   // Загружаем текущие флаги состояния
   #dm := #Bm;
   #Dx := #Bm;
   // Сбрасываем флаг первого цикла
   #Fx.Res := 0;
   // Назначаем группу сообщений (механизмов)
   // NDEV.GRP := SEL(G := 0 = #GRP, IN0 := #GRP, IN1 := PDEV.GRP);
   // Получаем структуру состояния привода
   IF (#Md.PZD) THEN
       #RRD := DPRD_DAT(LADDR := #LA, RECORD => #iT352);
   ELSE
       #RRD := DPRD_DAT(LADDR := #LA, RECORD => #iP6);
   END_IF;
   // Обрабатываем (непрерывные) данные состояния привода
   #SW := #SWx;
   #Re.X.SW := #SW;
   #Vx := #iT352.PZD2 / 16384.0 * #Vn;
   #Re.X.Vx := #Vx;
   #Ix := #iT352.PZD3 / 163.84;
   #Re.X.Ix := #Ix;
   #Mx := #iT352.PZD4 / 163.84;
   #Re.X.Mx := #Mx;
   #An := #iT352.PZD5;
   #Re.X.An := #An;
   #Fn := #iT352.PZD6;
   #Re.X.Fn := #Fn;
   #Brk := #iT352.PZD1.b02;
   #Re.X.Brk := #Brk;
   #Flt := #iT352.PZD1.b03 OR (#DPx = 0);
   #Re.X.Err := #Flt;
   #Alm := #iT352.PZD1.b07;
   // Обрабатываем дополнительные данные
   #P7 := #iT352.PZD7;
   #P8 := #iT352.PZD8;
   #P9 := #iT352.PZD9;
   // Передача параметров Master=>Slave
   IF (#Re.S.Mst) THEN
       // Данный привод является основным
       #Re."M".UBr := #UBr;
       #Re."M".Enb := #Enb;
       #Re."M".KOn := #KOn;
       #Re."M".Run := #Run;
       #Re."M".Ack := #Ack  OR "_ACK";
       #Re."M".Id := #Id;
       #Re."M".Ms := #Ms;
       #Re."M".Vs := #Vs;
       #Re."M".Vn := #Vn;
   ELSE
       // Данный привод является резервным
       #UBr := #Re."M".UBr;
       #Enb := #Re."M".Enb;
       #KOn := #Re."M".KOn;
       #Run := #Re."M".Run;
       #Ack := #Re."M".Ack;
       #Id := #Re."M".Id;
       #Ms := #Re."M".Ms;
       #Vs := #Re."M".Vs;
       #Vn := #Re."M".Vn;
   END_IF;
   // Формируем признаки устройства ввода резерва
   #Rd1 := #Re.S.Rd1;
   #SF.Rd1 := #Re.S.Rd1;
   #Rd2 := #Re.S.Rd2;
   #SF.Rd2 := #Re.S.Rd2;
   // Обработка состояния моторного модуля
   #SF.Flt := #Flt;
   #Fx.Flt := #Flt;
   #SF.Alm := #Alm;
   #Fx.Alm := #Alm;
   // Фиксируем текущие флаги
   #Fx.Mse :=  #Mse;               // (#PDEV.Msd = 0) &      // Разрешение выдачи сообщений для HMI
   #Fx.EnF := #Fx.Mse & #Md.EnF;                        // Разрешено сообщение Fault (отказ)
   #Fx.MsF := (#Fn <> 0) & #Fx.EnF;                        // Наличие сообщения Fault (отказ)
   #Fx.EnA := #Fx.Mse & #Md.EnA;                        // Разрешено сообщение Alarm (предупреждение)
   #Fx.MsA := (#An <> 0) & #Fx.EnA;                        // Наличие сообщения Alarm (предупреждение)
   #Fx.Rdy := #iT352.PZD1.b00;                         // Сигнал готовности привода (b00)
   #Fx.KOn := (#KOn OR #Run) & ((#Md.Rst = 0) OR #Fx.Rdy);  // Включить привод KOn|Run (команда)
   // Обрабатываем таймеры изменения состояния
   IF (#Fx.Tx0 OR #Fx.Tx1) THEN
       #Fx.Tx1 := ("_Time" - #Tm1 < #Ts1) & #Fx.Tx1;
       #Fx.Tx0 := ("_Time" - #Tm0 < #Md.Ts0) & #Fx.Tx0 & #Rdy & #Enb & (#Flt = 0);
   END_IF;
   // Фиксируем наличие событий
   #Dp := #Dx XOR #dm;
   // Обработка событий
   //  *** IF (#Dp <> 0) THEN
       // Запрос на инициализацию данных
   IF (#Fm.Res) THEN
           // Устанавливаем номер данного Instance Data Block
         (*#NDEV.IDB := 123; //- GetDINO();
           // Назначаем общие параметры сообщения
           #ME.Pr.N2 := #NDEV.IDB; *)
           // Инициализация данных
           #ME.Pr.N2 := 0;
           #ME.Pr.N4 := 0;
           #ME.Pr.N5 := 0;
           // Устанавливаем номер данного Instance Data Block
           #TPA := #ME;
           #NDB := #TSA.PTR.DN;
           // Назначаем группу сообщений (механизмов)
           IF (#GRP = 0) THEN
               #GRP := #NDB * 100;
           END_IF;
       END_IF;
       // Производим контроль изменения Rdy
       IF (#Fp.Rdy) THEN
           #Fx.Tx1 := (#Ts1 > T#0s) & #Fm.Rdy;
           #Tm1 := "_Time";
       END_IF;
       #Fx.Tx1 := (#Flt = 0) & #Fx.Tx1;
       #Rdy := #Fx.Tx1 OR #Fx.Rdy;
       #Re.X.Rdy := #Rdy;
       // Производим контроль изменения KOn
       IF (#Fp.KOn) THEN
           #Fx.Tx0 := (#Md.Ts0 > T#0s) & #Fm.KOn;
           #Tm0 := "_Time";
       END_IF;
       #Fx.Tx0 := (#Flt = 0) & #Fx.Tx0;
       #Fx.Run := #Fx.KOn OR #Fx.Tx0;
       // Устанавливаем активность сообщения Alarm (предупреждение)
       IF (#Fp.MsA XOR #MsAlm.SIG) THEN
           // Назначаем группу сообщений (механизмов)
           // Запрос на инициализацию данных
           #ME.Pr.N1 := #GRP;
           #ME.Pr.N2.%X0 := #Fm.MsA;
           #ME.Pr.N4 := 13;
           #ME.Pr.N6 := #GRP + 1;
           #MsAlm(SIG := (#Fp.MsA),
                  TIMESTAMP := "TS0",
                  SD_1 := #ME.Pr.N1,
                  SD_2 := #ME.Pr.N2,
                  SD_4 := #ME.Pr.N4,
                  SD_6 := #ME.Pr.N6);
       END_IF;
       // Устанавливаем активность сообщения Fault (отказ)
       IF (#Fp.MsF XOR #MsFlt.SIG)  THEN
          // Назначаем группу сообщений (механизмов)
          // Запрос на инициализацию данных
           #ME.Pr.N1 := #GRP;
           #ME.Pr.N2.%X0 := #Fm.MsF;
           #ME.Pr.N6 := #GRP + 2;
           #MsFlt(SIG := (#Fp.MsF),
                  TIMESTAMP := "TS0",
                  SD_1 := #ME.Pr.N1,
                  SD_2 := #ME.Pr.N2,
                  SD_6 := #ME.Pr.N6);
       END_IF;

       // Сохраняем текущее значение флагов
       #Bm := #Dx;
       //  *** END_IF;
   // Подготовка управляющей структуры привода
   #qT352.PZD1.b00 := ((#Re.S.Mst = 0) & #Re.S.Rd2 OR #Re.S.Mst & #Re.S.Rd1) & #Fx.Run;
   #qT352.PZD1.b02 := (#Re.S.Dis = 0) & #Enb & #DPx;
   #qT352.PZD1.b07 := #Re."M".Ack OR "_ACK";
   #qT352.PZD1.b12 := #UBr;
   // Обработка уставки скорости
   IF (#Run) THEN
       // Режим работы со скоростью и моментом
       #Vm := ABS(#Vn * 1.95);
       #Vs := LIMIT(MN := - #Vm, IN := #Vs, MX := + #Vm);
       #qT352.PZD2 := DINT_TO_INT(ROUND(#Vs / #Vn * 16384.0));
   ELSE
       // Режим намагничивания
       #qT352.PZD2 := 0;
   END_IF;
   // Обработка уставки момента
   IF (#Run OR #KOn) THEN
       #Ms := LIMIT(MN := -195.0, IN := #Ms, MX := +195.0);
       #qT352.PZD3 := DINT_TO_INT(ROUND(#Ms * 163.84));
   ELSE
       #qT352.PZD3 := 0;
   END_IF;
   // Формируем дополнительный параметр
   #qT352.PZD4 := #Id;
   // Передаем структуру управления привода
   IF (#Md.PZD) THEN
        #RWR := DPWR_DAT(LADDR := #LA, RECORD := #qT352);
   ELSE
        #RWR := DPWR_DAT(LADDR := #LA, RECORD := #qP6);
   END_IF;
   // Сбрасываем признак запрета
   #Re.S.Dis := 0;
   // Формируем индикацию для HMI
   #SF.Rdy := #Rdy;
   #SF.Qm0 := 0;
   #SF.Qm1 := #Re.S.Mst;
   #SF.Qm2 := #SF.Qm1 = 0;
END_FUNCTION_BLOCK

(* ===== HMI "HMI_RT_1" =====
system functions are stored by id; their names below are inferred from use
connection "HMI_Connection_1": ETHERNET, S7_1500_OMS

HMI tags "Default tag table"
   "Tag_ScreenNumber" : UInt, internal
   "AiCh_TE7.1_Px" : Real = PLC "AiCh_TE7.1".Px AT %DB7.DBD50, 1 s
   "AiCh_TE7.2_Px" : Real = PLC "AiCh_TE7.2".Px AT %DB8.DBD50, 1 s
   "Data_LevelVO_Pv" : Real = PLC Data.LevelVO_Pv, 1 s
   "DriveM7_1_Vx" : Real = PLC DriveM7_1.Vx AT %DB34.DBD78, 1 s
   "DriveM7_2_Vx" : Real = PLC DriveM7_2.Vx AT %DB35.DBD78, 1 s
   "AiCh_TE1.1_Px" : Real = PLC "AiCh_TE1.1".Px AT %DB1.DBD50, 1 s
   "AiCh_TE1.3_Px" : Real = PLC "AiCh_TE1.3".Px AT %DB3.DBD50, 1 s
   "AiCh_TE1.2_Px" : Real = PLC "AiCh_TE1.2".Px AT %DB2.DBD50, 1 s
   "DriveM1_1_Vx" : Real = PLC DriveM1_1.Vx AT %DB33.DBD78, 1 s
   "AiCh_LIC1.1_Px" : Real = PLC "AiCh_LIC1.1".Px AT %DB12.DBD50, 1 s
   "AiCh_TE2.1_Px" : Real = PLC "AiCh_TE2.1".Px AT %DB4.DBD50, 1 s
   "AiCh_TE2.3_Px" : Real = PLC "AiCh_TE2.3".Px AT %DB6.DBD50, 1 s
   "AiCh_TE2.2_Px" : Real = PLC "AiCh_TE2.2".Px AT %DB5.DBD50, 1 s
   "DriveM2_1_Vx" : Real = PLC DriveM2_1.Vx AT %DB38.DBD78, 1 s
   "AiCh_LIC2.1_Px" : Real = PLC "AiCh_LIC2.1".Px AT %DB13.DBD50, 1 s
   "Data_ACK" : Bool = PLC Data.Ack, 1 s
   "Data_MAN_ON" : Bool = PLC Data.MAN_ON, 1 s
   "Data_Reg_TE1_1_Sp" : Real = PLC Data.Reg_TE1_1.Sp, 1 s
   "Di_Lah1.1" : Bool = PLC "Di_Lah1.1" AT %I42.6, 1 s
   "Di_Ga1.4" : Bool = PLC "Di_Ga1.4" AT %I44.3, 1 s
   "DrvCell_M1_1_SB1" : Bool = PLC DrvCell_M1_1.SB1 AT %DB36.DBX16.0, 1 s
   "DrvCell_M1_1_Err" : Bool = PLC DrvCell_M1_1.Err AT %DB36.DBX74.1, 1 s
   "DrvCell_M1_1_Km1" : Bool = PLC DrvCell_M1_1.Km1 AT %DB36.DBX73.0, 1 s
   "DrvCell_M2_1_Err" : Bool = PLC DrvCell_M2_1.Err AT %DB37.DBX74.1, 1 s
   "DrvCell_M1_2_Km1" : Bool = PLC DrvCell_M1_2.Km1 AT %DB17.DBX73.0, 1 s
   "DrvCell_M1_2_Err" : Bool = PLC DrvCell_M1_2.Err AT %DB17.DBX74.1, 1 s
   "DrvCell_M1_2_SB1" : Bool = PLC DrvCell_M1_2.SB1 AT %DB17.DBX16.0, 1 s
   "DrvCell_V1_7_Err" : Bool = PLC DrvCell_V1_7.Err AT %DB28.DBX74.1, 1 s
   "DrvCell_V1_7_Km1" : Bool = PLC DrvCell_V1_7.Km1 AT %DB28.DBX73.0, 1 s
   "DrvCell_V1_7_SB1" : Bool = PLC DrvCell_V1_7.SB1 AT %DB28.DBX16.0, 1 s
   "Data_Mixer1_Direction" : Int = PLC Data.Mixer1.Direction, 1 s
   "Data_Equipment_Work" : Bool = PLC Data.Equipment_Work, 1 s
   "DrvCell_V1_1_SB1" : Bool = PLC DrvCell_V1_1.SB1 AT %DB25.DBX16.0, 1 s
   "DrvCell_V1_1_Err" : Bool = PLC DrvCell_V1_1.Err AT %DB25.DBX74.1, 1 s
   "DrvCell_M2_1_SB1" : Bool = PLC DrvCell_M2_1.SB1 AT %DB37.DBX16.0, 1 s
   "DrvCell_M2_1_Lr2" : Bool = PLC DrvCell_M2_1.Lr2 AT %DB37.DBX73.7, 1 s
   "DrvCell_M2_1_Km1" : Bool = PLC DrvCell_M2_1.Km1 AT %DB37.DBX73.0, 1 s
   "Data_Mixer2_Direction" : Int = PLC Data.Mixer2.Direction, 1 s
   "Di_Ga2.4" : Bool = PLC "Di_Ga2.4" AT %I44.7, 1 s
   "Data_Reg_TE2_1_Sp" : Real = PLC Data.Reg_TE2_1.Sp, 1 s
   "Di_Lah2.1" : Bool = PLC "Di_Lah2.1" AT %I42.7, 1 s
   "DrvCell_V2_1_SB1" : Bool = PLC DrvCell_V2_1.SB1 AT %DB26.DBX16.0, 1 s
   "DrvCell_V2_1_Err" : Bool = PLC DrvCell_V2_1.Err AT %DB26.DBX74.1, 1 s
   "DrvCell_V2_1_Km1" : Bool = PLC DrvCell_V2_1.Km1 AT %DB26.DBX73.0, 1 s
   "DrvCell_M2_2_SB1" : Bool = PLC DrvCell_M2_2.SB1 AT %DB18.DBX16.0, 1 s
   "DrvCell_M2_2_Err" : Bool = PLC DrvCell_M2_2.Err AT %DB18.DBX74.1, 1 s
   "DrvCell_M2_2_Km1" : Bool = PLC DrvCell_M2_2.Km1 AT %DB18.DBX73.0, 1 s
   "DrvCell_V2_7_SB1" : Bool = PLC DrvCell_V2_7.SB1 AT %DB29.DBX16.0, 1 s
   "DrvCell_V2_7_Err" : Bool = PLC DrvCell_V2_7.Err AT %DB29.DBX74.1, 1 s
   "DrvCell_V2_7_Km1" : Bool = PLC DrvCell_V2_7.Km1 AT %DB29.DBX73.0, 1 s
   "DrvCell_V1_1_Km1" : Bool = PLC DrvCell_V1_1.Km1 AT %DB25.DBX73.0, 1 s
   "Data_Mixer1_Man" : Real = PLC Data.Mixer1.Man, 1 s
   "Data_Mixer2_Man" : Real = PLC Data.Mixer2.Man, 1 s
   "Di_Ga1.1" : Bool = PLC "Di_Ga1.1" AT %I44.0, 1 s
   "Di_Ga1.2" : Bool = PLC "Di_Ga1.2" AT %I44.1, 1 s
   "Di_Ga2.1" : Bool = PLC "Di_Ga2.1" AT %I44.4, 1 s
   "Di_Ga2.2" : Bool = PLC "Di_Ga2.2" AT %I44.5, 1 s
   "DrvCell_M5_SB1" : Bool = PLC DrvCell_M5.SB1 AT %DB59.DBX16.0, 1 s
   "DrvCell_M5_Err" : Bool = PLC DrvCell_M5.Err AT %DB59.DBX74.1, 1 s
   "DrvCell_M5_Km1" : Bool = PLC DrvCell_M5.Km1 AT %DB59.DBX73.0, 1 s
   "DrvCell_M4_Err" : Bool = PLC DrvCell_M4.Err AT %DB21.DBX74.1, 1 s
   "DrvCell_M4_Km1" : Bool = PLC DrvCell_M4.Km1 AT %DB21.DBX73.0, 1 s
   "DrvCell_M4_SB1" : Bool = PLC DrvCell_M4.SB1 AT %DB21.DBX16.0, 1 s
   "Di_1Ga06" : Bool = PLC Di_1Ga06 AT %I46.4, 1 s
   "Di_1Ga01" : Bool = PLC Di_1Ga01 AT %I45.6, 1 s
   "Di_1Ga02" : Bool = PLC Di_1Ga02 AT %I46.0, 1 s
   "Data_Kr1_TempFilling" : Real = PLC Data.Kr1.TempFilling, 1 s
   "Data_Kr1_TempKristal" : Real = PLC Data.Kr1.TempKristal, 1 s
   "Kr_1_Work_Run" : Bool = PLC Kr_1_Work.Run, 1 s
   "Data_Kr1_TimeKristal" : Int = PLC Data.Kr1.TimeKristal, 1 s
   "Kr_1_Work_LeftTimeMin" : DInt = PLC Kr_1_Work.LeftTimeMin, 1 s
   "Data_Kr1_Regim" : Int = PLC Data.Kr1.Regim, 1 s
   "Data_Kr1_Start" : Bool = PLC Data.Kr1.Start, 1 s
   "Data_Kr1_Stop" : Bool = PLC Data.Kr1.Stop, 1 s
   "Data_Mixer1_Power" : Real = PLC Data.Mixer1.Power, 1 s
   "Data_Mixer1_TimeRight" : DInt = PLC Data.Mixer1.TimeRight, 1 s
   "Data_Mixer1_TimeLeft" : DInt = PLC Data.Mixer1.TimeLeft, 1 s
   "Data_Mixer1_TimePause" : DInt = PLC Data.Mixer1.TimePause, 1 s
   "Data_Mixer1_RegimBothSide" : Bool = PLC Data.Mixer1.RegimBothSide, 1 s
   "Data_Mixer1_Start" : Bool = PLC Data.Mixer1.Start, 1 s
   "Data_Mixer1_Stop" : Bool = PLC Data.Mixer1.Stop, 1 s
   "Data_Kr1_Ready_Work" : Bool = PLC Data.Kr1.Ready_Work, 1 s
   "Data_Kr1_Ready_Route" : Bool = PLC Data.Kr1.Ready_Route, 1 s
   "Data_GlobalErrorStop" : Bool = PLC Data.GlobalErrorStop, 1 s
   "Data_Kr2_TempFilling" : Real = PLC Data.Kr2.TempFilling, 1 s
   "Kr_2_Work_Run" : Bool = PLC Kr_2_Work.Run, 1 s
   "Data_Kr2_TempKristal" : Real = PLC Data.Kr2.TempKristal, 1 s
   "Data_Kr2_TimeKristal" : Int = PLC Data.Kr2.TimeKristal, 1 s
   "Kr_2_Work_LeftTimeMin" : DInt = PLC Kr_2_Work.LeftTimeMin, 1 s
   "Data_Kr2_Regim" : Int = PLC Data.Kr2.Regim, 1 s
   "Data_Kr2_Start" : Bool = PLC Data.Kr2.Start, 1 s
   "Data_Kr2_Stop" : Bool = PLC Data.Kr2.Stop, 1 s
   "Data_Kr2_Ready_Work" : Bool = PLC Data.Kr2.Ready_Work, 1 s
   "Data_Kr2_Ready_Route" : Bool = PLC Data.Kr2.Ready_Route, 1 s
   "Data_Mixer2_Power" : Real = PLC Data.Mixer2.Power, 1 s
   "Data_Mixer2_TimeRight" : DInt = PLC Data.Mixer2.TimeRight, 1 s
   "Data_Mixer2_TimeLeft" : DInt = PLC Data.Mixer2.TimeLeft, 1 s
   "Data_Mixer2_TimePause" : DInt = PLC Data.Mixer2.TimePause, 1 s
   "Data_Mixer2_RegimBothSide" : Bool = PLC Data.Mixer2.RegimBothSide, 1 s
   "Data_Mixer2_Start" : Bool = PLC Data.Mixer2.Start, 1 s
   "Data_Mixer2_Stop" : Bool = PLC Data.Mixer2.Stop, 1 s
   "Data_washing_cipRegim" : Int = PLC Data.washing.cipRegim, 1 s
   "Data_washing_Start" : Bool = PLC Data.washing.Start, 1 s
   "Data_washing_Stop" : Bool = PLC Data.washing.Stop, 1 s
   "Data_washing_readyGlobal" : Bool = PLC Data.washing.readyGlobal, 1 s
   "Data_washing_readyRoute" : Bool = PLC Data.washing.readyRoute, 1 s
   "WashingWork_DB_Run" : Bool = PLC WashingWork_DB.Run, 1 s
   "Data_Reg_M7_1_Sp" : Real = PLC Data.Reg_M7_1.Sp, 1 s
   "Data_Reg_01RV01_Sp" : Real = PLC Data.Reg_01RV01.Sp, 1 s
   "Data_Power_7_2" : Real = PLC Data.Power_7_2, 1 s
   "Kr_1_Work_Step" : Int = PLC Kr_1_Work.Step, 1 s
   "Kr_2_Work_Step" : Int = PLC Kr_2_Work.Step, 1 s
   "Data_GlobalError" : Bool = PLC Data.GlobalError, 1 s
   "DrvCell_V7_3_Err" : Bool = PLC DrvCell_V7_3.Err AT %DB31.DBX74.1, 1 s
   "DrvCell_V7_3_Km1" : Bool = PLC DrvCell_V7_3.Km1 AT %DB31.DBX73.0, 1 s
   "DrvCell_V7_4_Err" : Bool = PLC DrvCell_V7_4.Err AT %DB32.DBX74.1, 1 s
   "DrvCell_V7_4_Km1" : Bool = PLC DrvCell_V7_4.Km1 AT %DB32.DBX73.0, 1 s
   "DrvCell_V7_3_SB1" : Bool = PLC DrvCell_V7_3.SB1 AT %DB31.DBX16.0, 1 s
   "DrvCell_V7_4_SB1" : Bool = PLC DrvCell_V7_4.SB1 AT %DB32.DBX16.0, 1 s
   "Data_Reg_01RV01_LMN" : Real = PLC Data.Reg_01RV01.LMN, 1 s
   "Data_Reg_01RV01_Man" : Real = PLC Data.Reg_01RV01.Man, 1 s
   "DrvCell_V7_1_Err" : Bool = PLC DrvCell_V7_1.Err AT %DB23.DBX74.1, 1 s
   "DrvCell_V7_1_Km1" : Bool = PLC DrvCell_V7_1.Km1 AT %DB23.DBX73.0, 1 s
   "DrvCell_V7_1_SB1" : Bool = PLC DrvCell_V7_1.SB1 AT %DB23.DBX16.0, 1 s
   "DrvCell_M7_1_Err" : Bool = PLC DrvCell_M7_1.Err AT %DB39.DBX74.1, 1 s
   "DrvCell_M7_1_Km1" : Bool = PLC DrvCell_M7_1.Km1 AT %DB39.DBX73.0, 1 s
   "DrvCell_M7_1_SB1" : Bool = PLC DrvCell_M7_1.SB1 AT %DB39.DBX16.0, 1 s
   "Data_Reg_M7_1_Man" : Real = PLC Data.Reg_M7_1.Man, 1 s
   "DrvCell_M10_Err" : Bool = PLC DrvCell_M10.Err AT %DB22.DBX74.1, 1 s
   "DrvCell_M10_Km1" : Bool = PLC DrvCell_M10.Km1 AT %DB22.DBX73.0, 1 s
   "DrvCell_M10_SB1" : Bool = PLC DrvCell_M10.SB1 AT %DB22.DBX16.0, 1 s
   "DrvCell_M3_Err" : Bool = PLC DrvCell_M3.Err AT %DB20.DBX74.1, 1 s
   "DrvCell_M3_Km1" : Bool = PLC DrvCell_M3.Km1 AT %DB20.DBX73.0, 1 s
   "DrvCell_M3_SB1" : Bool = PLC DrvCell_M3.SB1 AT %DB20.DBX16.0, 1 s
   "Di_Lah01" : Bool = PLC Di_Lah01 AT %I43.1, 1 s
   "Di_Lal01" : Bool = PLC Di_Lal01 AT %I43.2, 1 s
   "DrvCell_M7_2_Err" : Bool = PLC DrvCell_M7_2.Err AT %DB40.DBX74.1, 1 s
   "DrvCell_M7_2_Km1" : Bool = PLC DrvCell_M7_2.Km1 AT %DB40.DBX73.0, 1 s
   "DrvCell_M7_2_SB1" : Bool = PLC DrvCell_M7_2.SB1 AT %DB40.DBX16.0, 1 s
   "Data_Reg_M7_2_Man" : Real = PLC Data.Reg_M7_2.Man, 1 s
   "DrvCell_V7_2_SB1" : Bool = PLC DrvCell_V7_2.SB1 AT %DB24.DBX16.0, 1 s
   "DrvCell_V7_2_Err" : Bool = PLC DrvCell_V7_2.Err AT %DB24.DBX74.1, 1 s
   "DrvCell_V7_2_Km1" : Bool = PLC DrvCell_V7_2.Km1 AT %DB24.DBX73.0, 1 s
   "ViewLine_DB_Line2" : Int = PLC ViewLine_DB.Line2, 1 s
   "ViewLine_DB_Line1" : Int = PLC ViewLine_DB.Line1, 1 s
   "ViewLine_DB_Line3" : Int = PLC ViewLine_DB.Line3, 1 s
   "ViewLine_DB_Line4" : Int = PLC ViewLine_DB.Line4, 1 s
   "ViewLine_DB_Line5" : Int = PLC ViewLine_DB.Line5, 1 s
   "ViewLine_DB_Line7" : Int = PLC ViewLine_DB.Line7, 1 s
   "ViewLine_DB_Line8" : Int = PLC ViewLine_DB.Line8, 1 s
   "ViewLine_DB_Line9" : Int = PLC ViewLine_DB.Line9, 1 s
   "ViewLine_DB_Line10" : Int = PLC ViewLine_DB.Line10, 1 s
   "ViewLine_DB_Line11" : Int = PLC ViewLine_DB.Line11, 1 s
   "ViewLine_DB_Line12" : Int = PLC ViewLine_DB.Line12, 1 s
   "Messages" : Word AT %DB44.DBW0, 1 s
   "ViewLine_DB_Line13" : Int = PLC ViewLine_DB.Line13, 1 s
   "ViewLine_DB_Line14" : Int = PLC ViewLine_DB.Line14, 1 s
   "ViewLine_DB_Line17" : Int = PLC ViewLine_DB.Line17, 1 s
   "ViewLine_DB_Line15" : Int = PLC ViewLine_DB.Line15, 1 s
   "ViewLine_DB_Line16" : Int = PLC ViewLine_DB.Line16, 1 s
   "ViewLine_DB_Line25" : Int = PLC ViewLine_DB.Line25, 1 s
   "ViewLine_DB_Line24" : Int = PLC ViewLine_DB.Line24, 1 s
   "ViewLine_DB_Line23" : Int = PLC ViewLine_DB.Line23, 1 s
   "ViewLine_DB_Line18" : Int = PLC ViewLine_DB.Line18, 1 s
   "ViewLine_DB_Line19" : Int = PLC ViewLine_DB.Line19, 1 s
   "ViewLine_DB_Line20" : Int = PLC ViewLine_DB.Line20, 1 s
   "ViewLine_DB_Line21" : Int = PLC ViewLine_DB.Line21, 1 s
   "ViewLine_DB_Line22" : Int = PLC ViewLine_DB.Line22, 1 s
   "WashingWork_DB_Step" : Int = PLC WashingWork_DB.Step, 1 s
   "Data_ReadyKr1" : Bool = PLC Data.ReadyKr1, 1 s
   "Data_Power_7_2_CIP" : Real = PLC Data.Power_7_2_CIP, 1 s
   "Data_EnableReady" : Bool = PLC Data.EnableReady, 1 s
   "Data_ReadyKr2" : Bool = PLC Data.ReadyKr2, 1 s
   "Data_ReadyCIP" : Bool = PLC Data.ReadyCIP, 1 s

discrete alarms
   11: 'Нажата аварийная кнопка', class Errors, trigger "Messages" bit 8
   12: 'Напряжение 380В не в норме', class Errors, trigger "Messages" bit 9
   13: 'Нет давления воздуха в пневмосистеме', class Errors, trigger "Messages" bit 10
   14: 'Верхний аварийный уровень кристализатора №1', class Errors, trigger "Messages" bit 11
   15: 'Верхний аварийный уровень кристализатора №2', class Errors, trigger "Messages" bit 12
   16: 'Верхний аварийный уровень емкости ледянной воды', class Errors, trigger "Messages" bit 13
   17: 'UPS, батарея разряжена', class Warnings, trigger "Messages" bit 14
   18: 'UPS, батарея неисправна', class No Acknowledgement, trigger "Messages" bit 15
   19: 'Открыт люк 1 кристализатора', class Errors, trigger "Messages" bit 0
   20: 'Открыт люк 2 кристализатора', class Errors, trigger "Messages" bit 1

text list "Kristal_Regim": 1 'Наполнение'; 2 'Кристализация'; 3 'Выкачка'

text list "cipRegim": 1 'Мойка линии подачи продукта'; 2 'Мойка линии выгрузки продукта'; 3 'Мойка кристализатора №1'; 4 'Мойка кристализатора №2'

text list "on/off": 0 'Отключено'; 1 'Включено'

Template "Template_1" 800x434
   Button "Template_Button_9" at 2,375 size 100x58; TextOff 'Вакуумный охладитель'
      on Release: ActivateScreen("mainVo", 0)
   AlarmView "Alarm view_Unacknowledged" at 0,357 size 800x19
   Button "Template_Button_5" at 104,375 size 100x58; TextOff 'Кристализа- торы'
      on Release: ActivateScreen("Kristals", 0)
   Button "Template_Button_6" at 406,375 size 96x58; TextOff 'Сообщения'
      on Release: ActivateScreen("messages", 0)
   Button "Template_Button_3" at 504,375 size 96x58; TextOff 'Настройки'
      on Release: ActivateScreen("SettingsCommon", 0)
   Button "Template_Button_4" at 206,375 size 100x58; TextOff 'Линии крист.'
      on Release: ActivateScreen("Lines", 0)
   Button "Template_Button_7" at 308,375 size 96x58; TextOff 'Графики'
      on Release: ActivateScreen("TrendsCommon", 0)
   Button "Template_Button_1" at 602,375 size 96x58; TextOff 'Сброс аварии'
      on Press: function_b14e0dd5("Data_ACK", 0)
   Button "Template_Button_2" at 700,375 size 96x58; TextOff 'Ручной'
      on Press: InvertBit("Data_MAN_ON")
      Appearance <- "Data_MAN_ON"
      ObjectEnable <- "Data_Equipment_Work"

screen "mainVo" 800x434, template "Template_1"
   on GenerateScreen: SetTag("Tag_ScreenNumber", 1)
   Rectangle "Rectangle_12" at 233,159 size 68x24; ToolTipText 'Температура НС'
   TextField "Text field_15" at 274,159 size 18x22; Text '%'
   IOField "IO Field_11" at 236,157 size 36x26; FormatPattern 999
      ProcessValue <- "Data_LevelVO_Pv"
   SymbolLibrary "Symbol library_35" at 261,235 size 13x60
      Appearance <- "ViewLine_DB_Line1"
   SymbolLibrary "Symbol library_56" at 167,48 size 13x149
      Appearance <- "ViewLine_DB_Line2"
   SymbolLibrary "Symbol library_1" at 63,195 size 166x13
      Appearance <- "ViewLine_DB_Line1"
   SymbolLibrary "Symbol library_6" at 255,12 size 54x54
   SymbolLibrary "Symbol library_9" at 217,28 size 25x25
      Appearance <- "ViewLine_DB_Line2"
   SymbolLibrary "Symbol library_4" at 219,39 size 98x199
   SymbolLibrary "Symbol library_31" at 714,259 size 13x43
      Appearance <- "DrvCell_M3_Km1"
   SymbolLibrary "Symbol library_160" at 714,143 size 13x49
   GraphicView "Graphic view_4" at 672,168 size 102x103; Picture "Graphic_5"
   SymbolLibrary "Symbol library_19" at 61,280 size 196x13
      Appearance <- "ViewLine_DB_Line7"
   SymbolLibrary "Symbol library_11" at 358,196 size 13x78
      Appearance <- "ViewLine_DB_Line7"
   SymbolLibrary "Symbol library_15" at 386,256 size 25x25
      Appearance <- "ViewLine_DB_Line3"
   SymbolLibrary "Symbol library_13" at 346,268 size 25x25
      Appearance <- "ViewLine_DB_Line7"
   Bar "Bar_1" at 223,67 size 90x143; MinimumValue 0; MaximumValue 100
      ProcessValue <- "Data_LevelVO_Pv"
   SymbolLibrary "Symbol library_7" at 307,12 size 55x28
   SymbolLibrary "Symbol library_2" at 188,28 size 37x13
      Appearance <- "ViewLine_DB_Line2"
   Group "Group_19" at 233,157 size 68x26
   SymbolLibrary "Symbol library_53" at 40,40 size 13x147
      Appearance <- "ViewLine_DB_Line1"
   SymbolLibrary "Symbol library_51" at 167,28 size 25x25
      Appearance <- "ViewLine_DB_Line2"
   SymbolLibrary "Symbol library_5" at 40,183 size 25x25
      Appearance <- "ViewLine_DB_Line1"
   SymbolLibrary "Symbol library_12" at 261,290 size 25x25
      Appearance <- "ViewLine_DB_Line1"
   SymbolLibrary "Symbol library_14" at 400,256 size 169x13
      Appearance <- "ViewLine_DB_Line3"
   SymbolLibrary "Symbol library_16" at 562,252 size 41x21
   SymbolLibrary "Symbol library_17" at 384,197 size 116x13
      Appearance <- "ViewLine_DB_Line5"
   SymbolLibrary "Symbol library_18" at 285,302 size 100x13
      Appearance <- "ViewLine_DB_Line1"
   SymbolLibrary "Symbol library_22" at 38,280 size 25x25
      Appearance <- "ViewLine_DB_Line7"
   SymbolLibrary "Symbol library_23" at 384,105 size 128x13
      Appearance <- "ViewLine_DB_Line4"
   SymbolLibrary "Symbol library_24" at 279,280 size 69x13
      Appearance <- "ViewLine_DB_Line7"
   SymbolLibrary "Symbol library_25" at 553,184 size 34x13
      Appearance <- "ViewLine_DB_Line5"
   TextField "Text field_2" at 592,205 size 23x43; Text 'Y'
   SymbolLibrary "Symbol library_29" at 507,67 size 25x25
      Appearance <- "ViewLine_DB_Line4"
   SymbolLibrary "Symbol library_30" at 585,184 size 25x25
      Appearance <- "ViewLine_DB_Line5"
   Circle "Circle_27" at 742,239 size 25x25
      Appearance <- "Di_Lal01"
   SymbolLibrary "Symbol library_36" at 702,299 size 25x25
      Appearance <- "DrvCell_M3_Km1"
   SymbolLibrary "Symbol library_34" at 613,296 size 61x13
      Appearance <- "DrvCell_M3_Km1"
   SymbolLibrary "Symbol library_161" at 591,292 size 25x21
   SymbolLibrary "Symbol library_37" at 710,122 size 21x25
   SymbolLibrary "Symbol library_27" at 531,67 size 113x13
      Appearance <- "ViewLine_DB_Line4"
   TextField "Static Text47_1" at 74,77 size 33x16; Text 'TE7.1 / TE04.1'
   Group "Group_17" at 49,91 size 82x26; FormatPattern 999.9
   SymbolLibrary "Symbol library_41" at 36,9 size 21x41
   TextField "Static Text47_2" at 176,213 size 33x16; Text 'TE7.2 / TE04.1'
   Group "Group_1" at 151,252 size 82x26; FormatPattern 999.9
   Group "Group_20" at 94,301 size 55x20; FormatPattern 999
   Group "Group_2" at 462,322 size 55x20; FormatPattern 999
   IOField "IO Field_12" at 36,243 size 47x31; FormatPattern 999
      Visibility <- "Data_MAN_ON"
      ProcessValue <- "Data_Reg_01RV01_Man"
   IOField "IO Field_2" at 466,287 size 47x31; FormatPattern 999
      Visibility <- "Data_MAN_ON"
      ProcessValue <- "Data_Reg_M7_1_Man"
   SymbolLibrary "Symbol library_20" at 258,340 size 108x7
      Appearance <- "ViewLine_DB_Line8"
   SymbolLibrary "Symbol library_42" at 241,336 size 30x15
   SymbolLibrary "Symbol library_44" at 362,334 size 15x13
      Appearance <- "ViewLine_DB_Line8"
   SymbolLibrary "Symbol library_43" at 369,316 size 15x13
      Appearance <- "ViewLine_DB_Line8"
   SymbolLibrary "Symbol library_45" at 412,143 size 81x7
      Appearance <- "ViewLine_DB_Line9"
   SymbolLibrary "Symbol library_47" at 400,138 size 30x15
   SymbolLibrary "Symbol library_49" at 490,137 size 11x13
      Appearance <- "ViewLine_DB_Line9"
   SymbolLibrary "Symbol library_50" at 494,118 size 12x13
      Appearance <- "ViewLine_DB_Line9"
   Group "Group_3" at 566,131 size 55x20; FormatPattern 999
   IOField "IO Field_3" at 570,92 size 47x31; FormatPattern 999
      Visibility <- "Data_MAN_ON"
      ProcessValue <- "Data_Reg_M7_2_Man"
   TextField "Text field_6" at 32,302 size 23x43; Text 'Y'
   TextField "Text field_7" at 647,87 size 23x43; Text 'Y'
   SymbolLibrary "Symbol library_28" at 640,67 size 25x25
      Appearance <- "ViewLine_DB_Line4"
   SymbolLibrary "Symbol library_38" at 494,130 size 7x14
      Appearance <- "ViewLine_DB_Line9"
   TextField "Static Text47_13" at 513,165 size 24x16; Text 'M10 / TE04.1'
   TextField "Static Text47_3" at 109,152 size 26x16; Text 'V7.3 / TE04.1'
   TextField "Static Text47_4" at 186,66 size 26x16; Text 'V7.4 / TE04.1'
   TextField "Static Text47_5" at 527,81 size 28x16; Text 'M7.2 / TE04.1'
   TextField "Static Text47_6" at 424,120 size 26x16; Text 'V7.2 / TE04.1'
   TextField "Static Text47_7" at 310,314 size 26x16; Text 'V7.1 / TE04.1'
   TextField "Static Text47_8" at 419,271 size 28x16; Text 'M7.1 / TE04.1'
   TextField "Static Text47_9" at 668,276 size 17x16; Text 'M3 / TE04.1'
   TextField "Static Text58_6" at 685,203 size 76x32; Text 'Ледянная вода RV01'
   Circle "Circle_26" at 742,176 size 25x25
      Appearance <- "Di_Lah01"
   ScreenModuleView "V7_31_1" at 105,169 size 43x40; ScreenModuleType ""
      Guid_{11997190-20001} <- "DrvCell_V7_3_Err"
      Guid_{11997190-19997} <- "DrvCell_V7_3_Km1"
   ScreenModuleView "M1_2_1" at 497,181 size 57x45; ScreenModuleType ""
      Guid_{11997190-21672} <- "DrvCell_M10_Err"
      Guid_{11997190-21676} <- "DrvCell_M10_Km1"
   ScreenModuleView "V1_7_1" at 308,330 size 30x25; ScreenModuleType ""
      Guid_{11997190-23352} <- "DrvCell_V7_1_Err"
      Guid_{11997190-23356} <- "DrvCell_V7_1_Km1"
   SymbolLibrary "Symbol library_3" at 341,8 size 44x222
   ScreenModuleView "RV01_2" at 87,234 size 51x64; ScreenModuleType ""
      Guid_{11997190-34850} <- "Data_Reg_01RV01_LMN"
   ScreenModuleView "М7_4_1" at 165,87 size 40x43; ScreenModuleType ""
      Guid_{11997190-20546} <- "DrvCell_V7_4_Err"
      Guid_{11997190-20554} <- "DrvCell_V7_4_Km1"
   Button "Button_6" at 85,148 size 73x73; TextOff 'Text'
      on Press: function_b14e0dd5("DrvCell_V7_3_SB1", 0)
   ScreenModuleView "M7_1_1" at 380,276 size 81x62; ScreenModuleType ""
      Guid_{11997190-20939} <- "DrvCell_M7_1_Err"
      Guid_{11997190-20935} <- "DrvCell_M7_1_Km1"
   Button "Button_7" at 374,242 size 88x113; TextOff 'Text'
      on Press: function_b14e0dd5("DrvCell_M7_1_SB1", 0)
   Button "Button_3" at 491,158 size 74x85; TextOff 'Text'
      on Press: function_b14e0dd5("DrvCell_M10_SB1", 0)
   ScreenModuleView "M_3_1" at 646,293 size 57x45; ScreenModuleType ""
      Guid_{11997190-24475} <- "DrvCell_M3_Err"
      Guid_{11997190-24471} <- "DrvCell_M3_Km1"
   Button "Button_8" at 637,271 size 74x85; TextOff 'Text'
      on Press: function_b14e0dd5("DrvCell_M3_SB1", 0)
   ScreenModuleView "V1_7_2" at 448,131 size 30x25; ScreenModuleType ""
      Guid_{11997190-23352} <- "DrvCell_V7_2_Err"
      Guid_{11997190-23356} <- "DrvCell_V7_2_Km1"
   ScreenModuleView "M7_21_1" at 504,91 size 59x53; ScreenModuleType ""
      Guid_{11997190-26153} <- "DrvCell_M7_2_Err"
      Guid_{11997190-26157} <- "DrvCell_M7_2_Km1"
   Group "Group_27" at 233,133 size 68x26
   Group "Group_4" at 151,228 size 82x26; FormatPattern 999.9
   Button "Button_1" at 494,67 size 74x85; TextOff 'Text'
      on Press: function_b14e0dd5("DrvCell_M7_2_SB1", 0)
   Button "Button_5" at 275,298 size 87x60; TextOff 'Text'
      on Press: function_b14e0dd5("DrvCell_V7_1_SB1", 0)
   Button "Button_2" at 414,115 size 74x53; TextOff 'Text'
      on Press: function_b14e0dd5("DrvCell_V7_2_SB1", 0)
   Button "Button_4" at 145,65 size 73x73; TextOff 'Text'
      on Press: function_b14e0dd5("DrvCell_V7_4_SB1", 0)
   SymbolLibrary "Symbol library_8" at 369,326 size 8x10
      Appearance <- "ViewLine_DB_Line8"
   Rectangle "Rectangle_1" at 56,93 size 75x24; ToolTipText 'Температура НС'
   TextField "Text field_3" at 106,93 size 19x22; Text 'С°'
   IOField "IO Field_10" at 49,91 size 56x26; FormatPattern 999.9
      ProcessValue <- "AiCh_TE7.1_Px"
   Rectangle "Rectangle_2" at 158,254 size 75x24; ToolTipText 'Температура НС'
   TextField "Text field_4" at 208,254 size 19x22; Text 'С°'
   IOField "IO Field_1" at 151,252 size 56x26; FormatPattern 999.9
      ProcessValue <- "AiCh_TE7.2_Px"
   IOField "I/O field_2" at 94,301 size 39x20; FormatPattern 999
      ProcessValue <- "Data_Reg_01RV01_LMN"
   TextField "Text field_16" at 130,302 size 19x19; Text '%'
   IOField "I/O field_1" at 462,322 size 39x20; FormatPattern 999
      ProcessValue <- "DriveM7_1_Vx"
   TextField "Text field_5" at 498,323 size 19x19; Text '%'
   IOField "I/O field_3" at 566,131 size 39x20; FormatPattern 999
      ProcessValue <- "DriveM7_2_Vx"
   TextField "Text field_1" at 602,132 size 19x19; Text '%'
   Rectangle "Rectangle_15" at 233,135 size 68x24; ToolTipText 'Температура НС'
   TextField "Text field_23" at 274,135 size 18x22; Text '%'
   IOField "IO Field_19" at 236,133 size 36x26; FormatPattern 999
      ProcessValue <- "Data_Reg_M7_1_Sp"
   Rectangle "Rectangle_3" at 158,230 size 75x24; ToolTipText 'Температура НС'
   TextField "Text field_8" at 208,230 size 19x22; Text 'С°'
   IOField "IO Field_4" at 151,228 size 56x26; FormatPattern 999.9
      ProcessValue <- "Data_Reg_01RV01_Sp"

screen "TrendsCommon" 800x434, template "Template_1"
   Button "Template_Button_7g" at 256,50 size 308x58; TextOff 'Вакуумохладитель'
      on Release: ActivateScreen("VO", 0)
   Button "Template_Button_8" at 256,109 size 308x58; TextOff 'Кристализатор №1'
      on Release: ActivateScreen("Kristalizator1", 0)
   Button "Template_Button_10" at 256,168 size 308x58; TextOff 'Кристализатор №2'
      on Release: ActivateScreen("Kristalizator2", 0)

screen "messages" 800x434, template "Template_1"
   AlarmView "Alarm view_1" at 0,2 size 798x321
   Button "Template_Button_5q" at 618,323 size 82x34; TextOff 'Архив'
      on Release: ActivateScreen("messagesArchive", 0)

screen "messagesArchive" 800x434, template "Template_1"
   AlarmView "Alarm view_1" at 0,0 size 798x356; AlarmLog "Alarm_log_1"

screen "VO" 800x434, template "Template_1"
   TrendView "Trend view_1" at 0,0 size 798x356

screen "Kristalizator1" 800x434, template "Template_1"
   TrendView "Trend view_1" at 0,0 size 798x356

screen "Kristalizator2" 800x434, template "Template_1"
   TrendView "Trend view_1" at 0,0 size 798x356

screen "Kristals" 800x434, template "Template_1"
   SymbolLibrary "Symbol library_164" at 144,10 size 41x32
      Visibility <- "Data_Mixer1_Direction"
   SymbolLibrary "Symbol library_126" at 260,10 size 41x32
      Visibility <- "Data_Mixer1_Direction"
   Rectangle "Rectangle_6" at 47,93 size 75x24; ToolTipText 'Температура НС'
   IOField "IO Field_5" at 40,91 size 56x26; FormatPattern 999.9
      ProcessValue <- "AiCh_TE1.2_Px"
   TextField "Text field_9" at 97,93 size 19x22; Text 'С°'
   Group "Group_14" at 40,91 size 82x26
   TextField "Static Text47_7" at 63,75 size 36x17; Text 'TE1.2 / TE04.1'
   SymbolLibrary "Symbol library_1" at 230,326 size 76x13
      Appearance <- "ViewLine_DB_Line13"
   SymbolLibrary "Symbol library_66" at 161,266 size 25x25
      Appearance <- "ViewLine_DB_Line11"
   GraphicView "Graphic view_5" at 147,60 size 154x223; Picture "Graphic_1"
   Bar "Bar_2" at 170,76 size 110x191; MinimumValue 0; MaximumValue 100
      ProcessValue <- "AiCh_LIC1.1_Px"
   SymbolLibrary "Symbol library_17" at 188,67 size 72x113
   TextField "Text field_7" at 161,90 size 55x39; Text '№1'
   ScreenModuleView "M1_1_1" at 194,0 size 53x69; ScreenModuleType ""
      Guid_{11997190-22971} <- "DrvCell_M1_1_Err"
      Guid_{11997190-22975} <- "DrvCell_M1_1_Km1"
   SymbolLibrary "Symbol library_59" at 78,313 size 72x13
      Appearance <- "ViewLine_DB_Line12"
   SymbolLibrary "Symbol library_63" at 181,290 size 25x25
      Appearance <- "ViewLine_DB_Line11"
   SymbolLibrary "Symbol library_64" at 134,110 size 13x205
      Appearance <- "ViewLine_DB_Line11"
   SymbolLibrary "Symbol library_67" at 134,100 size 25x25
      Appearance <- "ViewLine_DB_Line11"
   SymbolLibrary "Symbol library_68" at 58,309 size 25x21
   SymbolLibrary "Symbol library_147" at 110,122 size 25x25
      Appearance <- "ViewLine_DB_Line11"
   SymbolLibrary "Symbol library_148" at 107,141 size 21x25
   SymbolLibrary "Symbol library_65" at 181,278 size 25x25
      Appearance <- "ViewLine_DB_Line11"
   SymbolLibrary "Symbol library_44" at 219,308 size 13x45
      Appearance <- "ViewLine_DB_Line10"
   SymbolLibrary "Symbol library_57" at 215,277 size 31x42
   SymbolLibrary "Symbol library_50" at 299,322 size 24x21
   TextField "Static Text47_8" at 90,222 size 33x16; Text 'TE1.3 / TE04.1'
   Group "Group_10" at 65,236 size 82x26
   TextField "Static Text47_9" at 306,108 size 40x16; Text 'LIC 1.1 / TE04.1'
   TextField "Static Text47_6" at 206,182 size 33x16; Text 'TE1.1 / TE04.1'
   Group "Group_7" at 181,220 size 82x26
   Group "Group_26" at 181,196 size 82x26; FormatPattern 999.9
   Circle "Circle_23" at 295,72 size 25x25
      Appearance <- "Di_Lah1.1"
   SymbolLibrary "Symbol library_2" at 275,10 size 89x13
      Appearance <- "ViewLine_DB_Line24"
   SymbolLibrary "Symbol library_3" at 258,33 size 13x59
      Appearance <- "ViewLine_DB_Line24"
   SymbolLibrary "Symbol library_4" at 352,7 size 24x21
   SymbolLibrary "Symbol library_5" at 258,10 size 25x25
      Appearance <- "ViewLine_DB_Line24"
   Rectangle "Rectangle_17" at 180,71 size 19x18
      Appearance <- "Di_Ga1.4"
   ScreenModuleView "V7_31_1" at 90,287 size 43x40; ScreenModuleType ""
      Guid_{11997190-20001} <- "DrvCell_V1_1_Err"
      Guid_{11997190-19997} <- "DrvCell_V1_1_Km1"
   TextField "Static Text47_18" at 92,271 size 26x16; Text 'V1.1 / TE04.1'
   TextField "Static Text47_1" at 183,329 size 28x16; Text 'M1.2 / TE04.1'
   ScreenModuleView "V1_7_1" at 257,316 size 30x25; ScreenModuleType ""
      Guid_{11997190-23352} <- "DrvCell_V1_7_Err"
      Guid_{11997190-23356} <- "DrvCell_V1_7_Km1"
   TextField "Static Text47_2" at 259,298 size 26x16; Text 'V1.7 / TE04.1'
   TextField "Static Text58_1" at 381,8 size 45x16; Text 'CIP+1 / RV01'
   SymbolLibrary "Symbol library_6" at 579,326 size 76x13
      Appearance <- "ViewLine_DB_Line17"
   SymbolLibrary "Symbol library_7" at 510,266 size 25x25
      Appearance <- "ViewLine_DB_Line15"
   GraphicView "Graphic view_1" at 496,60 size 154x223; Picture "Graphic_1"
   Bar "Bar_1" at 519,76 size 110x191; MinimumValue 0; MaximumValue 100
      ProcessValue <- "AiCh_LIC2.1_Px"
   SymbolLibrary "Symbol library_8" at 537,67 size 72x113
   TextField "Text field_1" at 510,90 size 55x39; Text '№2'
   ScreenModuleView "M1_1_2" at 543,0 size 53x69; ScreenModuleType ""
      Guid_{11997190-22971} <- "DrvCell_M2_1_Err"
      Guid_{11997190-22975} <- "DrvCell_M2_1_Km1"
   SymbolLibrary "Symbol library_9" at 427,313 size 73x13
   SymbolLibrary "Symbol library_10" at 530,290 size 25x25
      Appearance <- "ViewLine_DB_Line15"
   SymbolLibrary "Symbol library_11" at 483,110 size 13x205
      Appearance <- "ViewLine_DB_Line15"
   SymbolLibrary "Symbol library_12" at 483,100 size 25x25
      Appearance <- "ViewLine_DB_Line15"
   SymbolLibrary "Symbol library_13" at 406,309 size 25x21
      Appearance <- "ViewLine_DB_Line16"
   SymbolLibrary "Symbol library_14" at 459,122 size 25x25
      Appearance <- "ViewLine_DB_Line15"
   SymbolLibrary "Symbol library_15" at 456,141 size 21x25
   SymbolLibrary "Symbol library_16" at 530,278 size 25x25
      Appearance <- "ViewLine_DB_Line15"
   SymbolLibrary "Symbol library_18" at 568,308 size 13x45
      Appearance <- "ViewLine_DB_Line14"
   SymbolLibrary "Symbol library_19" at 564,277 size 31x42
   SymbolLibrary "Symbol library_20" at 648,322 size 24x21
   TextField "Static Text47_4" at 439,222 size 33x16; Text 'TE2.3 / TE04.1'
   Group "Group_3" at 414,236 size 82x26
   TextField "Static Text47_5" at 655,108 size 40x16; Text 'LIC 2.1 / TE04.1'
   TextField "Static Text47_10" at 555,182 size 33x16; Text 'TE2.1 / TE04.1'
   Group "Group_5" at 530,220 size 82x26
   Group "Group_8" at 530,196 size 82x26; FormatPattern 999.9
   Circle "Circle_1" at 644,72 size 25x25
      Appearance <- "Di_Lah2.1"
   SymbolLibrary "Symbol library_21" at 624,10 size 89x13
      Appearance <- "ViewLine_DB_Line25"
   SymbolLibrary "Symbol library_22" at 607,33 size 13x59
      Appearance <- "ViewLine_DB_Line25"
   SymbolLibrary "Symbol library_23" at 701,7 size 24x21
   SymbolLibrary "Symbol library_24" at 607,10 size 25x25
      Appearance <- "ViewLine_DB_Line25"
   Rectangle "Rectangle_10" at 529,71 size 19x18
      Appearance <- "Di_Ga2.4"
   ScreenModuleView "V7_31_2" at 438,287 size 43x40; ScreenModuleType ""
      Guid_{11997190-20001} <- "DrvCell_V2_1_Err"
      Guid_{11997190-19997} <- "DrvCell_V2_1_Km1"
   TextField "Static Text47_11" at 438,271 size 26x16; Text 'V2.1 / TE04.1'
   TextField "Static Text47_12" at 532,329 size 28x16; Text 'M2.2 / TE04.1'
   ScreenModuleView "V1_7_2" at 606,316 size 30x25; ScreenModuleType ""
      Guid_{11997190-23352} <- "DrvCell_V2_7_Err"
      Guid_{11997190-23356} <- "DrvCell_V2_7_Km1"
   TextField "Static Text47_13" at 608,298 size 26x16; Text 'V2.7 / TE04.1'
   TextField "Static Text58_2" at 730,8 size 45x16; Text 'CIP+1 / RV01'
   Button "Button_2" at 596,295 size 65x56; TextOff 'Text'
      on Press: function_b14e0dd5("DrvCell_V2_7_SB1", 0)
   Group "Group_6" at 294,122 size 68x26
   Group "Group_4" at 643,122 size 68x26
   IOField "IO Field_15" at 84,6 size 51x31; FormatPattern s999
      Visibility <- "Data_MAN_ON"
      ProcessValue <- "Data_Mixer1_Man"
   IOField "IO Field_10" at 436,6 size 51x31; FormatPattern s999
      Visibility <- "Data_MAN_ON"
      ProcessValue <- "Data_Mixer2_Man"
   Button "Button_4" at 409,279 size 73x73; TextOff 'Text'
      on Press: function_b14e0dd5("DrvCell_V2_1_SB1", 0)
   Group "Group_23" at 109,47 size 63x20; FormatPattern 999
   Group "Group_15" at 40,75 size 82x42
   Group "Group_2" at 387,75 size 82x42
   Group "Group_11" at 459,47 size 63x20; FormatPattern 999
   SymbolLibrary "Symbol library_27" at 134,301 size 25x25
      Appearance <- "ViewLine_DB_Line11"
   ScreenModuleView "M1_2_1" at 147,300 size 46x37; ScreenModuleType ""
      Guid_{11997190-21676} <- "DrvCell_M1_2_Km1"
      Guid_{11997190-21672} <- "DrvCell_M1_2_Err"
   Button "Button_11" at 247,295 size 65x56; TextOff 'Text'
      on Press: function_b14e0dd5("DrvCell_V1_7_SB1", 0)
   SymbolLibrary "Symbol library_28" at 483,301 size 25x25
      Appearance <- "ViewLine_DB_Line15"
   ScreenModuleView "M1_2_2" at 496,300 size 46x37; ScreenModuleType ""
      Guid_{11997190-21672} <- "DrvCell_M2_2_Err"
      Guid_{11997190-21676} <- "DrvCell_M2_2_Km1"
   Button "Button_6" at 60,279 size 73x73; TextOff 'Text'
      on Press: function_b14e0dd5("DrvCell_V1_1_SB1", 0)
   Button "Button_12" at 177,1 size 105x78; TextOff 'Text'
      on Press: function_b14e0dd5("DrvCell_M1_1_SB1", 0)
   Group "Group" at 144,10 size 157x32
   Button "Button_3" at 526,1 size 105x78; TextOff 'Text'
      on Press: function_b14e0dd5("DrvCell_M2_1_SB1", 0)
   Group "Group_9" at 493,10 size 157x32
   Button "Button_1" at 491,278 size 70x74; TextOff 'Text'
      on Press: function_b14e0dd5("DrvCell_M2_2_SB1", 0)
   Button "Button_10" at 140,278 size 70x74; TextOff 'Text'
      on Press: function_b14e0dd5("DrvCell_M1_2_SB1", 0)
   Rectangle "Rectangle_5" at 72,238 size 75x24; ToolTipText 'Температура НС'
   IOField "IO Field_4" at 65,236 size 56x26; FormatPattern 999.9
      ProcessValue <- "AiCh_TE1.3_Px"
   TextField "Text field_8" at 122,238 size 19x22; Text 'С°'
   Rectangle "Rectangle_4" at 294,124 size 68x24; ToolTipText 'Температура НС'
   TextField "Text field_6" at 335,124 size 18x22; Text '%'
   IOField "IO Field_3" at 297,122 size 36x26; FormatPattern 999
      ProcessValue <- "AiCh_LIC1.1_Px"
   Rectangle "Rectangle_3" at 188,222 size 75x24; ToolTipText 'Температура НС'
   TextField "Text field_4" at 238,222 size 19x22; Text 'С°'
   IOField "IO Field_2" at 181,220 size 56x26; FormatPattern 999.9
      ProcessValue <- "AiCh_TE1.1_Px"
   Rectangle "Rectangle_14" at 188,198 size 75x24; ToolTipText 'Температура НС'
   TextField "Text field_22" at 238,198 size 19x22; Text 'С°'
   IOField "IO Field_18" at 181,196 size 56x26; FormatPattern 999.9
      ProcessValue <- "Data_Reg_TE1_1_Sp"
   Rectangle "Rectangle_1" at 394,93 size 75x24; ToolTipText 'Температура НС'
   IOField "IO Field_1" at 387,91 size 56x26; FormatPattern 999.9
      ProcessValue <- "AiCh_TE2.2_Px"
   TextField "Text field_2" at 444,93 size 19x22; Text 'С°'
   Group "Group_1" at 387,91 size 82x26
   TextField "Static Text47_3" at 410,75 size 36x17; Text 'TE2.2 / TE04.1'
   Rectangle "Rectangle_2" at 421,238 size 75x24; ToolTipText 'Температура НС'
   IOField "IO Field_6" at 414,236 size 56x26; FormatPattern 999.9
      ProcessValue <- "AiCh_TE2.3_Px"
   TextField "Text field_3" at 471,238 size 19x22; Text 'С°'
   Rectangle "Rectangle_7" at 643,124 size 68x24; ToolTipText 'Температура НС'
   TextField "Text field_5" at 684,124 size 18x22; Text '%'
   IOField "IO Field_7" at 646,122 size 36x26; FormatPattern 999
      ProcessValue <- "AiCh_LIC2.1_Px"
   Rectangle "Rectangle_8" at 537,222 size 75x24; ToolTipText 'Температура НС'
   TextField "Text field_10" at 587,222 size 19x22; Text 'С°'
   IOField "IO Field_8" at 530,220 size 56x26; FormatPattern 999.9
      ProcessValue <- "AiCh_TE2.1_Px"
   Rectangle "Rectangle_9" at 537,198 size 75x24; ToolTipText 'Температура НС'
   TextField "Text field_11" at 587,198 size 19x22; Text 'С°'
   IOField "IO Field_9" at 530,196 size 56x26; FormatPattern 999.9
      ProcessValue <- "Data_Reg_TE2_1_Sp"
   SymbolLibrary "Symbol library_25" at 493,10 size 41x32
      Visibility <- "Data_Mixer2_Direction"
   SymbolLibrary "Symbol library_26" at 609,10 size 41x32
      Visibility <- "Data_Mixer2_Direction"
   IOField "I/O field_4" at 109,47 size 43x20; FormatPattern s999
      ProcessValue <- "DriveM1_1_Vx"
   TextField "Text field_19" at 153,48 size 19x19; Text '%'
   IOField "I/O field_1" at 459,47 size 43x20; FormatPattern s999
      ProcessValue <- "DriveM2_1_Vx"
   TextField "Text field_12" at 503,48 size 19x19; Text '%'

screen "Lines" 800x434, template "Template_1"
   SymbolLibrary "Symbol library_33" at 545,38 size 25x25
      Visibility <- "Di_1Ga01"
      Appearance <- "ViewLine_DB_Line24"
   SymbolLibrary "Symbol library_31" at 511,50 size 43x13
      Visibility <- "Di_1Ga01"
      Appearance <- "ViewLine_DB_Line24"
   SymbolLibrary "Symbol library_32" at 557,28 size 13x24
      Visibility <- "Di_1Ga01"
      Appearance <- "ViewLine_DB_Line24"
   SymbolLibrary "Symbol library_34" at 545,66 size 25x25
      Visibility <- "Di_1Ga02"
      Appearance <- "ViewLine_DB_Line25"
   SymbolLibrary "Symbol library_35" at 510,78 size 43x13
      Visibility <- "Di_1Ga02"
      Appearance <- "ViewLine_DB_Line25"
   SymbolLibrary "Symbol library_36" at 557,36 size 13x44
      Visibility <- "Di_1Ga02"
      Appearance <- "ViewLine_DB_Line25"
   Rectangle "Rectangle_4" at 155,168 size 68x24; ToolTipText 'Температура НС'
   TextField "Text field_6" at 196,168 size 18x22; Text '%'
   IOField "IO Field_3" at 158,166 size 36x26; FormatPattern 999
      ProcessValue <- "AiCh_LIC1.1_Px"
   Rectangle "Rectangle_1" at 302,168 size 68x24; ToolTipText 'Температура НС'
   TextField "Text field_5" at 343,168 size 18x22; Text '%'
   IOField "IO Field_7" at 305,166 size 36x26; FormatPattern 999
      ProcessValue <- "AiCh_LIC2.1_Px"
   SymbolLibrary "Symbol library_40" at 93,315 size 47x13
      Appearance <- "ViewLine_DB_Line23"
   SymbolLibrary "Symbol library_39" at 139,315 size 148x13
      Appearance <- "ViewLine_DB_Line18"
   SymbolLibrary "Symbol library_21" at 547,178 size 71x13
      Appearance <- "ViewLine_DB_Line21"
   SymbolLibrary "Symbol library_90" at 93,22 size 414x13
      Appearance <- "ViewLine_DB_Line23"
   SymbolLibrary "Symbol library_64" at 77,46 size 13x260
      Appearance <- "ViewLine_DB_Line23"
   SymbolLibrary "Symbol library_67" at 77,22 size 25x25
      Appearance <- "ViewLine_DB_Line23"
   SymbolLibrary "Symbol library_1" at 77,303 size 25x25
      Appearance <- "ViewLine_DB_Line23"
   SymbolLibrary "Symbol library_2" at 289,315 size 173x13
      Appearance <- "ViewLine_DB_Line19"
   SymbolLibrary "Symbol library_3" at 102,248 size 77x13
      Appearance <- "ViewLine_DB_Line3"
   TextField "Static Text58_1" at 471,245 size 40x16; Text 'CIP-2 / RV01'
   SymbolLibrary "Symbol library_6" at 24,248 size 44x13
      Appearance <- "ViewLine_DB_Line3"
   SymbolLibrary "Symbol library_7" at 7,244 size 24x21
   TextField "Static Text58_2" at 1,201 size 71x32; Text 'Продукт, CIP+2 RV01'
   SymbolLibrary "Symbol library_8" at 184,157 size 13x129
      Appearance <- "ViewLine_DB_Line10"
   SymbolLibrary "Symbol library_5" at 330,157 size 13x129
      Appearance <- "ViewLine_DB_Line14"
   SymbolLibrary "Symbol library_9" at 509,302 size 24x13
      Appearance <- "ViewLine_DB_Line20"
   SymbolLibrary "Symbol library_10" at 536,143 size 13x156
      Appearance <- "ViewLine_DB_Line20"
   SymbolLibrary "Symbol library_11" at 524,290 size 25x25
      Appearance <- "ViewLine_DB_Line20"
   SymbolLibrary "Symbol library_12" at 547,120 size 102x13
      Appearance <- "ViewLine_DB_Line20"
   SymbolLibrary "Symbol library_13" at 536,120 size 24x25
      Appearance <- "ViewLine_DB_Line20"
   SymbolLibrary "Symbol library_14" at 637,115 size 24x21
   TextField "Static Text58_4" at 663,109 size 71x32; Text 'Продукт, CIP+1 RV01'
   SymbolLibrary "Symbol library_15" at 769,32 size 13x262
      Appearance <- "ViewLine_DB_Line22"
   SymbolLibrary "Symbol library_17" at 624,303 size 25x25
      Appearance <- "ViewLine_DB_Line21"
   SymbolLibrary "Symbol library_16" at 646,315 size 49x13
      Appearance <- "ViewLine_DB_Line21"
   SymbolLibrary "Symbol library_18" at 757,290 size 25x25
      Appearance <- "ViewLine_DB_Line22"
   SymbolLibrary "Symbol library_19" at 570,22 size 198x13
      Appearance <- "ViewLine_DB_Line22"
   SymbolLibrary "Symbol library_20" at 757,22 size 25x25
      Appearance <- "ViewLine_DB_Line22"
   SymbolLibrary "Symbol library_22" at 612,178 size 25x25
      Appearance <- "ViewLine_DB_Line21"
   SymbolLibrary "Symbol library_23" at 624,192 size 13x25
      Appearance <- "ViewLine_DB_Line21"
   GraphicView "Graphic view_2" at 583,205 size 94x103; Picture "Graphic_5"
   TextField "Static Text58_3" at 617,233 size 25x32; Text 'CIP ББ RV01'
   TextField "Static Text47_28" at 482,280 size 17x16; Text 'M5 / TE04.1'
   SymbolLibrary "Symbol library_25" at 735,302 size 34x13
      Appearance <- "ViewLine_DB_Line22"
   TextField "Static Text47_1" at 715,280 size 17x16; Text 'M4 / TE04.1'
   SymbolLibrary "Symbol library_26" at 203,248 size 122x13
      Appearance <- "ViewLine_DB_Line3"
   SymbolLibrary "Symbol library_27" at 348,248 size 108x13
      Appearance <- "ViewLine_DB_Line3"
   SymbolLibrary "Symbol library_4" at 444,244 size 24x21
   Line "Line_3" at 147,255 size 42x26
      Visibility <- "Di_Ga1.1"
   Line "Line_1" at 147,283 size 42x36
      Visibility <- "Di_Ga1.2"
   Line "Line_5" at 292,255 size 42x26
      Visibility <- "Di_Ga2.1"
   Line "Line_6" at 293,283 size 42x36
      Visibility <- "Di_Ga2.2"
   ScreenModuleView "M1_2_1" at 692,299 size 53x44; ScreenModuleType ""
      Guid_{11997190-21672} <- "DrvCell_M4_Err"
      Guid_{11997190-21676} <- "DrvCell_M4_Km1"
   ScreenModuleView "M1_2_2" at 459,299 size 53x44; ScreenModuleType ""
      Guid_{11997190-21672} <- "DrvCell_M5_Err"
      Guid_{11997190-21676} <- "DrvCell_M5_Km1"
   SymbolLibrary "Symbol library_24" at 217,50 size 286x13
      Appearance <- "ViewLine_DB_Line24"
   SymbolLibrary "Symbol library_94" at 511,22 size 50x13
      Visibility <- "Di_1Ga06"
      Appearance <- "ViewLine_DB_Line23"
   Group "Group" at 511,28 size 59x35
   Group "Group_1" at 510,36 size 60x55
   GraphicView "Graphic view_5" at 139,77 size 100x141; Picture "Graphic_1"
   Bar "Bar_2" at 152,91 size 75x117; MinimumValue 0; MaximumValue 100
      ProcessValue <- "AiCh_LIC1.1_Px"
   GraphicView "Graphic view_1" at 286,77 size 100x141; Picture "Graphic_1"
   Bar "Bar_1" at 299,91 size 75x117; MinimumValue 0; MaximumValue 100
      ProcessValue <- "AiCh_LIC2.1_Px"
   SymbolLibrary "Symbol library_29" at 203,66 size 13x37
      Appearance <- "ViewLine_DB_Line24"
   SymbolLibrary "Symbol library_28" at 364,78 size 139x13
      Appearance <- "ViewLine_DB_Line25"
   SymbolLibrary "Symbol library_30" at 203,50 size 25x25
      Appearance <- "ViewLine_DB_Line24"
   SymbolLibrary "Symbol library_37" at 353,78 size 25x25
      Appearance <- "ViewLine_DB_Line25"
   TextField "Static Text47_9" at 167,152 size 40x16; Text 'LIC 1.1 / TE04.1'
   Group "Group_6" at 155,166 size 68x26
   TextField "Static Text47_5" at 314,152 size 40x16; Text 'LIC 2.1 / TE04.1'
   Group "Group_4" at 302,166 size 68x26
   TextField "Text field_7" at 146,98 size 44x31; Text '№1'
   TextField "Text field_1" at 295,98 size 44x31; Text '№2'
   SymbolLibrary "Symbol library_57" at 182,215 size 24x30
   SymbolLibrary "Symbol library_38" at 328,215 size 24x30
   Button "Button_10" at 444,270 size 88x87; TextOff 'Text'
      on Press: function_b14e0dd5("DrvCell_M5_SB1", 0)
   Button "Button_1" at 676,273 size 88x87; TextOff 'Text'
      on Press: function_b14e0dd5("DrvCell_M4_SB1", 0)

screen "KR_1" 800x434, template "Template_1"
   TextField "Template_Text field_7" at 22,6 size 376x29; Text 'Параметры кристализации №1'
   IOField "IO Field_4" at 340,36 size 60x36; FormatPattern 999.9
      ProcessValue <- "Data_Kr1_TempFilling"
      ObjectEnable <- "Kr_1_Work_Run"
   TextField "Template_Text field_8" at 17,42 size 234x25; Text 'Температура наполнения, С°'
   IOField "IO Field_5" at 340,73 size 60x36; FormatPattern 999.9
      ProcessValue <- "Data_Kr1_TempKristal"
      ObjectEnable <- "Kr_1_Work_Run"
   TextField "Template_Text field_9" at 17,79 size 257x25; Text 'Температура кристализации, С°'
   IOField "IO Field_6" at 340,110 size 60x36; FormatPattern 9999
      ObjectEnable <- "Kr_1_Work_Run"
      ProcessValue <- "Data_Kr1_TimeKristal"
   TextField "Template_Text field_10" at 22,116 size 217x25; Text 'Время кристализации, мин'
   IOField "IO Field_7" at 340,147 size 60x36; FormatPattern 999
      ProcessValue <- "Kr_1_Work_LeftTimeMin"
   TextField "Template_Text field_11" at 22,153 size 241x25; Text 'До конца кристализации, мин'
   SymbolicIOField "Symbolic I/O field_kr1" at 22,185 size 378x55; TextOn '1'; TextOff '0'; TextList "Kristal_Regim"
      ObjectEnable <- "Kr_1_Work_Run"
      ProcessValue <- "Data_Kr1_Regim"
   Button "Button_2123" at 22,243 size 183x48; TextOff 'Старт'
      on Press: function_b14e0dd5("Data_Kr1_Start", 0)
   Button "Button_1123" at 217,243 size 183x48; TextOff 'Стоп'
      on Press: function_b14e0dd5("Data_Kr1_Stop", 0)
   TextField "Template_Text field_1" at 457,6 size 302x29; Text 'Параметры мешалки №1'
   IOField "IO Field_15" at 724,35 size 60x40; FormatPattern 999
      ProcessValue <- "Data_Mixer1_Power"
   TextField "Template_Text field_2" at 424,43 size 174x25; Text 'Обороты мешалки, %'
   IOField "IO Field_1" at 724,76 size 60x40; FormatPattern 9999
      ProcessValue <- "Data_Mixer1_TimeRight"
   TextField "Template_Text field_3" at 424,84 size 231x25; Text 'Время вращения вправо, сек'
   IOField "IO Field_2" at 724,117 size 60x40; FormatPattern 9999
      ProcessValue <- "Data_Mixer1_TimeLeft"
   TextField "Template_Text field_4" at 424,125 size 221x25; Text 'Время вращения влево, сек'
   IOField "IO Field_3" at 724,158 size 60x40; FormatPattern 9999
      ProcessValue <- "Data_Mixer1_TimePause"
   TextField "Template_Text field_5" at 424,166 size 179x25; Text 'Время паузы мешалки'
   TextField "Template_Text field_6" at 424,217 size 130x25; Text 'Режим мешалки'
   Button "Button_9" at 569,206 size 105x46; TextOff '<< || >>'
      on Release: SetBit("Data_Mixer1_RegimBothSide")
      Appearance <- "Data_Mixer1_RegimBothSide"
   Button "Button_10" at 679,206 size 105x46; TextOff '>>'
      on Release: ResetBit("Data_Mixer1_RegimBothSide")
      Appearance <- "Data_Mixer1_RegimBothSide"
   Button "Template_Button_1z" at 423,278 size 177x51; TextOff 'Старт мешалки'
      on Press: function_b14e0dd5("Data_Mixer1_Start", 0)
   Button "Template_Button_2q" at 607,278 size 177x51; TextOff 'Стоп мешалки'
      on Press: function_b14e0dd5("Data_Mixer1_Stop", 0)
   Circle "Circle_1" at 137,297 size 24x24
      Appearance <- "Data_Kr1_Ready_Work"
   TextField "Template_Text field_12" at 165,296 size 93x25; Text 'Готовность'
   Circle "Circle_2" at 21,330 size 20x20
      Appearance <- "Data_Kr1_Ready_Route"
   TextField "Template_Text field_13" at 45,328 size 74x25; Text 'Маршрут'
   Circle "Circle_3" at 138,330 size 20x20
      Appearance <- "Data_MAN_ON"
   TextField "Template_Text field_14" at 165,328 size 70x25; Text 'Автомат'
   Circle "Circle_4" at 249,330 size 20x20
      Appearance <- "Data_ReadyKr1"
   TextField "Template_Text field_15" at 272,328 size 100x25; Text 'Разрешение'

screen "KR_2" 800x434, template "Template_1"
   TextField "Template_Text field_7" at 22,6 size 376x29; Text 'Параметры кристализации №2'
   IOField "IO Field_4" at 340,36 size 60x36; FormatPattern 999.9
      ProcessValue <- "Data_Kr2_TempFilling"
      ObjectEnable <- "Kr_2_Work_Run"
   TextField "Template_Text field_8" at 17,42 size 234x25; Text 'Температура наполнения, С°'
   IOField "IO Field_5" at 340,73 size 60x36; FormatPattern 999.9
      ProcessValue <- "Data_Kr2_TempKristal"
      ObjectEnable <- "Kr_2_Work_Run"
   TextField "Template_Text field_9" at 17,79 size 257x25; Text 'Температура кристализации, С°'
   IOField "IO Field_6" at 340,110 size 60x36; FormatPattern 9999
      ProcessValue <- "Data_Kr2_TimeKristal"
      ObjectEnable <- "Kr_2_Work_Run"
   TextField "Template_Text field_10" at 22,116 size 217x25; Text 'Время кристализации, мин'
   IOField "IO Field_7" at 340,147 size 60x36; FormatPattern 999
      ProcessValue <- "Kr_2_Work_LeftTimeMin"
   TextField "Template_Text field_11" at 22,153 size 241x25; Text 'До конца кристализации, мин'
   SymbolicIOField "Symbolic I/O field_kr1" at 22,185 size 378x55; TextOn '1'; TextOff '0'; TextList "Kristal_Regim"
      ProcessValue <- "Data_Kr2_Regim"
      ObjectEnable <- "Kr_2_Work_Run"
   Button "Button_2123" at 22,243 size 183x48; TextOff 'Старт'
      on Press: function_b14e0dd5("Data_Kr2_Start", 0)
   Button "Button_1123" at 217,243 size 183x48; TextOff 'Стоп'
      on Press: function_b14e0dd5("Data_Kr2_Stop", 0)
   TextField "Template_Text field_1" at 457,6 size 302x29; Text 'Параметры мешалки №2'
   IOField "IO Field_15" at 724,35 size 60x40; FormatPattern 999
      ProcessValue <- "Data_Mixer2_Power"
   TextField "Template_Text field_2" at 424,43 size 174x25; Text 'Обороты мешалки, %'
   IOField "IO Field_1" at 724,76 size 60x40; FormatPattern 9999
      ProcessValue <- "Data_Mixer2_TimeRight"
   TextField "Template_Text field_3" at 424,84 size 231x25; Text 'Время вращения вправо, сек'
   IOField "IO Field_2" at 724,117 size 60x40; FormatPattern 9999
      ProcessValue <- "Data_Mixer2_TimeLeft"
   TextField "Template_Text field_4" at 424,125 size 221x25; Text 'Время вращения влево, сек'
   IOField "IO Field_3" at 724,158 size 60x40; FormatPattern 9999
      ProcessValue <- "Data_Mixer2_TimePause"
   TextField "Template_Text field_5" at 424,166 size 179x25; Text 'Время паузы мешалки'
   TextField "Template_Text field_6" at 424,217 size 130x25; Text 'Режим мешалки'
   Button "Button_9" at 569,206 size 105x46; TextOff '<< || >>'
      on Release: SetBit("Data_Mixer2_RegimBothSide")
      Appearance <- "Data_Mixer2_RegimBothSide"
   Button "Button_10" at 679,206 size 105x46; TextOff '>>'
      on Release: ResetBit("Data_Mixer2_RegimBothSide")
      Appearance <- "Data_Mixer2_RegimBothSide"
   Button "Template_Button_1z" at 423,278 size 177x51; TextOff 'Старт мешалки'
      on Press: function_b14e0dd5("Data_Mixer2_Start", 0)
   Button "Template_Button_2q" at 607,278 size 177x51; TextOff 'Стоп мешалки'
      on Press: function_b14e0dd5("Data_Mixer2_Stop", 0)
   Circle "Circle_1" at 137,297 size 24x24
      Appearance <- "Data_Kr2_Ready_Work"
   TextField "Template_Text field_12" at 165,296 size 93x25; Text 'Готовность'
   Circle "Circle_2" at 21,330 size 20x20
      Appearance <- "Data_Kr2_Ready_Route"
   TextField "Template_Text field_13" at 45,328 size 74x25; Text 'Маршрут'
   Circle "Circle_3" at 138,330 size 20x20
      Appearance <- "Data_MAN_ON"
   TextField "Template_Text field_14" at 165,328 size 70x25; Text 'Автомат'
   Circle "Circle_4" at 249,330 size 20x20
      Appearance <- "Data_ReadyKr2"
   TextField "Template_Text field_15" at 272,328 size 100x25; Text 'Разрешение'

screen "SettingsCommon" 800x434, template "Template_1"
   Button "Template_Button_7e" at 256,50 size 308x58; TextOff 'Кристализатор №1'
      on Release: ActivateScreen("KR_1", 0)
   Button "Template_Button_8" at 256,109 size 308x58; TextOff 'Кристализатор №2'
      on Release: ActivateScreen("KR_2", 0)
   Button "Template_Button_10" at 256,168 size 308x58; TextOff 'CIP мойка'
      on Release: ActivateScreen("CIP", 0)
   Button "Template_Button_1xz" at 256,227 size 308x58; TextOff 'Общие настройки'
      on Release: ActivateScreen("SetValue", 0)

screen "SetValue" 800x434, template "Template_1"
   TextField "Template_Text field_7" at 304,6 size 217x29; Text 'Общие настройки'
   IOField "IO Field_4" at 541,42 size 60x36; FormatPattern 999.9
      ProcessValue <- "Data_Reg_M7_1_Sp"
   TextField "Template_Text field_8" at 203,48 size 244x25; Text 'Уровень вакуумохладителя, %'
   IOField "IO Field_1" at 541,91 size 60x36; FormatPattern 999.9
      ProcessValue <- "Data_Reg_01RV01_Sp"
   TextField "Template_Text field_1" at 203,86 size 231x46; Text 'Температура продукта после вакуумного охладителя, C°'
   IOField "IO Field_2" at 541,139 size 60x36; FormatPattern 999.9
      ProcessValue <- "Data_Power_7_2"
   TextField "Template_Text field_2" at 203,145 size 313x25; Text 'Мощность насоса M7_2 на продукте, %'
   IOField "IO Field_3" at 541,184 size 60x36; FormatPattern 999.9
      ProcessValue <- "Data_Power_7_2_CIP"
   TextField "Template_Text field_3" at 203,190 size 290x25; Text 'Мощность насоса M7_2 на мойке, %'
   TextField "Template_Text field_4" at 203,233 size 310x25; Text 'Блокировка разрешение на включение'
   SymbolicIOField "Symbolic I/O field_1" at 203,266 size 182x42; TextOn '1'; TextOff '0'; Authorization "Operate"; TextList "on/off"
      ProcessValue <- "Data_EnableReady"

screen "CIP" 800x434, template "Template_1"
   TextField "Template_Text field_7" at 266,6 size 292x29; Text 'Управление CIP мойкой'
   SymbolicIOField "Symbolic I/O field_kr1" at 195,50 size 431x55; TextOn '1'; TextOff '0'; TextList "cipRegim"
      ProcessValue <- "Data_washing_cipRegim"
      ObjectEnable <- "WashingWork_DB_Run"
   Button "Button_2123" at 195,108 size 204x55; TextOff 'Старт'
      on Press: function_b14e0dd5("Data_washing_Start", 0)
   Button "Button_1123" at 422,108 size 204x55; TextOff 'Стоп'
      on Press: function_b14e0dd5("Data_washing_Stop", 0)
   Circle "Circle_1" at 320,192 size 28x28
      Appearance <- "Data_washing_readyGlobal"
   TextField "Template_Text field_12" at 356,194 size 93x25; Text 'Готовность'
   Circle "Circle_2" at 348,228 size 24x24
      Appearance <- "Data_washing_readyRoute"
   TextField "Template_Text field_1" at 383,226 size 74x25; Text 'Маршрут'
   Circle "Circle_3" at 348,263 size 24x24
      Appearance <- "Data_MAN_ON"
   TextField "Template_Text field_2" at 383,261 size 70x25; Text 'Автомат'
   Circle "Circle_4" at 348,298 size 24x24
      Appearance <- "Data_ReadyCIP"
   TextField "Template_Text field_3" at 383,296 size 100x25; Text 'Разрешение'
*)

(* ===== HMI "HMI_RT_3" =====
system functions are stored by id; their names below are inferred from use
connection "HMI_Connection_2": ETHERNET, S7_1500_OMS

HMI tags "Default tag table"
   "Di_1Ga06" : Bool = PLC Di_1Ga06 AT %I46.4, 1 s
   "AiCh_LIC1.1_Px" : Real = PLC "AiCh_LIC1.1".Px AT %DB12.DBD50, 1 s
   "Di_Ga3.3" : Bool = PLC "Di_Ga3.3" AT %I45.2, 1 s
   "AiCh_TE7.1_Px" : Real = PLC "AiCh_TE7.1".Px AT %DB7.DBD50, 1 s
   "AiCh_LIC7.2_Px" : Real = PLC "AiCh_LIC7.2".Px AT %DB16.DBD50, 1 s
   "DrvCell_M7_1_Km1" : Bool = PLC DrvCell_M7_1.Km1 AT %DB39.DBX73.0, 1 s
   "DrvCell_M7_1_Err" : Bool = PLC DrvCell_M7_1.Err AT %DB39.DBX74.1, 1 s
   "AiCh_TE1.1_Px" : Real = PLC "AiCh_TE1.1".Px AT %DB1.DBD50, 1 s
   "DrvCell_M1_1_Err" : Bool = PLC DrvCell_M1_1.Err AT %DB36.DBX74.1, 1 s
   "DrvCell_M1_1_Km1" : Bool = PLC DrvCell_M1_1.Km1 AT %DB36.DBX73.0, 1 s
   "AiCh_TE1.3_Px" : Real = PLC "AiCh_TE1.3".Px AT %DB3.DBD50, 1 s
   "AiCh_TE1.2_Px" : Real = PLC "AiCh_TE1.2".Px AT %DB2.DBD50, 1 s
   "Tag_ScreenNumber" : Int AT %DB1.DBX0.0
   "DrvCell_V7_3_Err" : Bool = PLC DrvCell_V7_3.Err AT %DB31.DBX74.1, 1 s
   "DrvCell_V7_3_Km1" : Bool = PLC DrvCell_V7_3.Km1 AT %DB31.DBX73.0, 1 s
   "DrvCell_V7_3_SB1" : Bool = PLC DrvCell_V7_3.SB1 AT %DB31.DBX16.0, 1 s
   "DrvCell_V7_4_Err" : Bool = PLC DrvCell_V7_4.Err AT %DB32.DBX74.1, 1 s
   "DrvCell_V7_4_Km1" : Bool = PLC DrvCell_V7_4.Km1 AT %DB32.DBX73.0, 1 s
   "DrvCell_V7_4_SB1" : Bool = PLC DrvCell_V7_4.SB1 AT %DB32.DBX16.0, 1 s
   "DrvCell_M10_Km1" : Bool = PLC DrvCell_M10.Km1 AT %DB22.DBX73.0, 1 s
   "DrvCell_M10_Err" : Bool = PLC DrvCell_M10.Err AT %DB22.DBX74.1, 1 s
   "DrvCell_M10_SB1" : Bool = PLC DrvCell_M10.SB1 AT %DB22.DBX16.0, 1 s
   "DrvCell_M3_Err" : Bool = PLC DrvCell_M3.Err AT %DB20.DBX74.1, 1 s
   "DrvCell_M3_Km1" : Bool = PLC DrvCell_M3.Km1 AT %DB20.DBX73.0, 1 s
   "DrvCell_M3_2_SB1" : Bool = PLC DrvCell_M3_2.SB1 AT %DB19.DBX16.0, 1 s
   "DrvCell_M7_2_Err" : Bool = PLC DrvCell_M7_2.Err AT %DB40.DBX74.1, 1 s
   "DrvCell_M7_2_Km1" : Bool = PLC DrvCell_M7_2.Km1 AT %DB40.DBX73.0, 1 s
   "DrvCell_M7_1_SB1" : Bool = PLC DrvCell_M7_1.SB1 AT %DB39.DBX16.0, 1 s
   "DrvCell_M7_2_SB1" : Bool = PLC DrvCell_M7_2.SB1 AT %DB40.DBX16.0, 1 s
   "DrvCell_V7_1_Err" : Bool = PLC DrvCell_V7_1.Err AT %DB23.DBX74.1, 1 s
   "DrvCell_V7_1_Km1" : Bool = PLC DrvCell_V7_1.Km1 AT %DB23.DBX73.0, 1 s
   "DrvCell_V7_1_SB1" : Bool = PLC DrvCell_V7_1.SB1 AT %DB23.DBX16.0, 1 s
   "DrvCell_V7_2_Err" : Bool = PLC DrvCell_V7_2.Err AT %DB24.DBX74.1, 1 s
   "DrvCell_V7_2_Km1" : Bool = PLC DrvCell_V7_2.Km1 AT %DB24.DBX73.0, 1 s
   "DrvCell_V7_2_SB1" : Bool = PLC DrvCell_V7_2.SB1 AT %DB24.DBX16.0, 1 s
   "DrvCell_V1_1_Err" : Bool = PLC DrvCell_V1_1.Err AT %DB25.DBX74.1, 1 s
   "DrvCell_V1_1_Km1" : Bool = PLC DrvCell_V1_1.Km1 AT %DB25.DBX73.0, 1 s
   "DrvCell_V1_1_SB1" : Bool = PLC DrvCell_V1_1.SB1 AT %DB25.DBX16.0, 1 s
   "DrvCell_M1_2_Err" : Bool = PLC DrvCell_M1_2.Err AT %DB17.DBX74.1, 1 s
   "DrvCell_M1_2_Km1" : Bool = PLC DrvCell_M1_2.Km1 AT %DB17.DBX73.0, 1 s
   "DrvCell_M1_2_SB1" : Bool = PLC DrvCell_M1_2.SB1 AT %DB17.DBX16.0, 1 s
   "DrvCell_V1_7_Err" : Bool = PLC DrvCell_V1_7.Err AT %DB28.DBX74.1, 1 s
   "DrvCell_V1_7_Km1" : Bool = PLC DrvCell_V1_7.Km1 AT %DB28.DBX73.0, 1 s
   "DrvCell_V1_7_SB1" : Bool = PLC DrvCell_V1_7.SB1 AT %DB28.DBX16.0, 1 s
   "DrvCell_M1_1_SB1" : Bool = PLC DrvCell_M1_1.SB1 AT %DB36.DBX16.0, 1 s
   "DrvCell_M2_1_Err" : Bool = PLC DrvCell_M2_1.Err AT %DB37.DBX74.1, 1 s
   "DrvCell_M2_1_Km1" : Bool = PLC DrvCell_M2_1.Km1 AT %DB37.DBX73.0, 1 s
   "DrvCell_M2_1_SB1" : Bool = PLC DrvCell_M2_1.SB1 AT %DB37.DBX16.0, 1 s
   "DrvCell_M2_2_Err" : Bool = PLC DrvCell_M2_2.Err AT %DB18.DBX74.1, 1 s
   "DrvCell_M2_2_Km1" : Bool = PLC DrvCell_M2_2.Km1 AT %DB18.DBX73.0, 1 s
   "DrvCell_M2_2_SB1" : Bool = PLC DrvCell_M2_2.SB1 AT %DB18.DBX16.0, 1 s
   "DrvCell_V2_7_Err" : Bool = PLC DrvCell_V2_7.Err AT %DB29.DBX74.1, 1 s
   "DrvCell_V2_7_Km1" : Bool = PLC DrvCell_V2_7.Km1 AT %DB29.DBX73.0, 1 s
   "DrvCell_V2_7_SB1" : Bool = PLC DrvCell_V2_7.SB1 AT %DB29.DBX16.0, 1 s
   "DrvCell_M4_Err" : Bool = PLC DrvCell_M4.Err AT %DB21.DBX74.1, 1 s
   "DrvCell_M4_Km1" : Bool = PLC DrvCell_M4.Km1 AT %DB21.DBX73.0, 1 s
   "DrvCell_M4_SB1" : Bool = PLC DrvCell_M4.SB1 AT %DB21.DBX16.0, 1 s
   "AiCh_TE2.2_Px" : Real = PLC "AiCh_TE2.2".Px AT %DB5.DBD50, 1 s
   "AiCh_TE2.3_Px" : Real = PLC "AiCh_TE2.3".Px AT %DB6.DBD50, 1 s
   "AiCh_TE2.1_Px" : Real = PLC "AiCh_TE2.1".Px AT %DB4.DBD50, 1 s
   "AiCh_LIC2.1_Px" : Real = PLC "AiCh_LIC2.1".Px AT %DB13.DBD50, 1 s
   "Di_Lah1.1" : Bool = PLC "Di_Lah1.1" AT %I42.6, 1 s
   "Di_Lah2.1" : Bool = PLC "Di_Lah2.1" AT %I42.7, 1 s
   "Di_Lah01" : Bool = PLC Di_Lah01 AT %I43.1, 1 s
   "Di_Lal01" : Bool = PLC Di_Lal01 AT %I43.2, 1 s
   "Di_Ga1.1" : Bool = PLC "Di_Ga1.1" AT %I44.0, 1 s
   "Di_Ga1.2" : Bool = PLC "Di_Ga1.2" AT %I44.1, 1 s
   "Di_Ga1.3" : Bool = PLC "Di_Ga1.3" AT %I44.2, 1 s
   "Di_Ga2.1" : Bool = PLC "Di_Ga2.1" AT %I44.4, 1 s
   "Di_Ga2.2" : Bool = PLC "Di_Ga2.2" AT %I44.5, 1 s
   "Di_Ga2.3" : Bool = PLC "Di_Ga2.3" AT %I44.6, 1 s
   "Di_1Ga01" : Bool = PLC Di_1Ga01 AT %I45.6, 1 s
   "Di_1Ga02" : Bool = PLC Di_1Ga02 AT %I46.0, 1 s
   "AiCh_TE7.2_Px" : Real = PLC "AiCh_TE7.2".Px AT %DB8.DBD50, 1 s
   "DriveM1_1.Vx" : Real = PLC DriveM1_1.Vx AT %DB33.DBD78, 1 s
   "DriveM2_1.Vx" : Real = PLC DriveM2_1.Vx AT %DB38.DBD78, 1 s
   "DriveM7_1.Vx" : Real = PLC DriveM7_1.Vx AT %DB34.DBD78, 1 s
   "DriveM7_2.Vx" : Real = PLC DriveM7_2.Vx AT %DB35.DBD78, 1 s
   "Data_ACK" : Bool = PLC Data.Ack, 1 s
   "Messages" : Word AT %DB44.DBW0, 1 s
   "Data_Reg_01RV01_LMN" : Real = PLC Data.Reg_01RV01.LMN, 1 s
   "Data_Mixer1_Power" : Real = PLC Data.Mixer1.Power, 1 s
   "Data_Mixer1_TimeRight" : DInt = PLC Data.Mixer1.TimeRight, 1 s
   "Data_Mixer1_TimeLeft" : DInt = PLC Data.Mixer1.TimeLeft, 1 s
   "Data_Mixer1_TimePause" : DInt = PLC Data.Mixer1.TimePause, 1 s
   "Data_Mixer1_RegimBothSide" : Bool = PLC Data.Mixer1.RegimBothSide, 1 s
   "Data_Mixer2_Power" : Real = PLC Data.Mixer2.Power, 1 s
   "Data_Mixer2_TimeRight" : DInt = PLC Data.Mixer2.TimeRight, 1 s
   "Data_Mixer2_TimeLeft" : DInt = PLC Data.Mixer2.TimeLeft, 1 s
   "Data_Mixer2_TimePause" : DInt = PLC Data.Mixer2.TimePause, 1 s
   "Data_Mixer2_RegimBothSide" : Bool = PLC Data.Mixer2.RegimBothSide, 1 s
   "DrvCell_V2_1_Err" : Bool = PLC DrvCell_V2_1.Err AT %DB26.DBX74.1, 1 s
   "DrvCell_V2_1_Km1" : Bool = PLC DrvCell_V2_1.Km1 AT %DB26.DBX73.0, 1 s
   "Data_MAN_ON" : Bool = PLC Data.MAN_ON, 1 s
   "DrvCell_M3_SB1" : Bool = PLC DrvCell_M3.SB1 AT %DB20.DBX16.0, 1 s
   "DrvCell_V2_1_SB1" : Bool = PLC DrvCell_V2_1.SB1 AT %DB26.DBX16.0, 1 s
   "Data_Reg_01RV01_Man" : Real = PLC Data.Reg_01RV01.Man, 1 s
   "Data_Reg_M7_1_Man" : Real = PLC Data.Reg_M7_1.Man, 1 s
   "Data_Reg_M7_2_Man" : Real = PLC Data.Reg_M7_2.Man, 1 s
   "Data_Mixer1_Man" : Real = PLC Data.Mixer1.Man, 1 s
   "Data_Mixer2_Man" : Real = PLC Data.Mixer2.Man, 1 s
   "Data_washing_readyGlobal" : Bool = PLC Data.washing.readyGlobal, 1 s
   "Data_washing_readyRoute" : Bool = PLC Data.washing.readyRoute, 1 s
   "Data_GlobalError" : Bool = PLC Data.GlobalError, 1 s
   "Data_washing_cipRegim" : Int = PLC Data.washing.cipRegim, 1 s
   "Data_washing_Start" : Bool = PLC Data.washing.Start, 1 s
   "Data_washing_Stop" : Bool = PLC Data.washing.Stop, 1 s
   "DrvCell_M5_Err" : Bool = PLC DrvCell_M5.Err AT %DB59.DBX74.1, 1 s
   "DrvCell_M5_Km1" : Bool = PLC DrvCell_M5.Km1 AT %DB59.DBX73.0, 1 s
   "DrvCell_M5_SB1" : Bool = PLC DrvCell_M5.SB1 AT %DB59.DBX16.0, 1 s
   "Data.LevelVO" : Real = PLC Data.LevelVO_Pv AT %DB1.DBW0, 1 s
   "Data_Kr1_TempFilling" : Real = PLC Data.Kr1.TempFilling, 1 s
   "Data_Kr1_TempKristal" : Real = PLC Data.Kr1.TempKristal, 1 s
   "Data_Kr1_TimeKristal" : Int = PLC Data.Kr1.TimeKristal, 1 s
   "Data_Mixer1_Start" : Bool = PLC Data.Mixer1.Start, 1 s
   "Data_Mixer1_Stop" : Bool = PLC Data.Mixer1.Stop, 1 s
   "Data_Mixer1_Direction" : Int = PLC Data.Mixer1.Direction, 1 s
   "Data_Mixer2_Direction" : Int = PLC Data.Mixer2.Direction, 1 s
   "Data_Mixer2_Start" : Bool = PLC Data.Mixer2.Start, 1 s
   "Data_Mixer2_Stop" : Bool = PLC Data.Mixer2.Stop, 1 s
   "Data_Reg_01RV01_Sp" : Real = PLC Data.Reg_01RV01.Sp, 1 s
   "Data_Reg_TE1_1_Sp" : Real = PLC Data.Reg_TE1_1.Sp, 1 s
   "Data_Reg_M7_1_LMN" : Real = PLC Data.Reg_M7_1.LMN, 1 s
   "Data_Kr1_Regim" : Int = PLC Data.Kr1.Regim, 1 s
   "Data_Kr1_Start" : Bool = PLC Data.Kr1.Start, 1 s
   "Data_Kr1_Stop" : Bool = PLC Data.Kr1.Stop, 1 s
   "Data_Kr1_Ready_Work" : Bool = PLC Data.Kr1.Ready_Work, 1 s
   "Data_Kr1_Ready_Route" : Bool = PLC Data.Kr1.Ready_Route, 1 s
   "Data_Reg_M7_2_LMN" : Real = PLC Data.Reg_M7_2.LMN, 1 s
   "Kr_1_Work_LeftTimeMin" : DInt = PLC Kr_1_Work.LeftTimeMin, 1 s
   "Kr_1_Work_TempHour" : Real = PLC Kr_1_Work.TempHour, 1 s
   "Data_Kr2_TempFilling" : Real = PLC Data.Kr2.TempFilling, 1 s
   "Data_Kr2_TempKristal" : Real = PLC Data.Kr2.TempKristal, 1 s
   "Data_Kr2_TimeKristal" : Int = PLC Data.Kr2.TimeKristal, 1 s
   "Kr_2_Work_LeftTimeMin" : DInt = PLC Kr_2_Work.LeftTimeMin, 1 s
   "Kr_2_Work_TempHour" : Real = PLC Kr_2_Work.TempHour, 1 s
   "Data_Kr2_Regim" : Int = PLC Data.Kr2.Regim, 1 s
   "Data_Kr2_Start" : Bool = PLC Data.Kr2.Start, 1 s
   "Data_Kr2_Stop" : Bool = PLC Data.Kr2.Stop, 1 s
   "Data_Kr2_Ready_Work" : Bool = PLC Data.Kr2.Ready_Work, 1 s
   "Data_Kr2_Ready_Route" : Bool = PLC Data.Kr2.Ready_Route, 1 s
   "Data_Reg_TE2_1_Sp" : Real = PLC Data.Reg_TE2_1.Sp, 1 s
   "Di_Ga1.4" : Bool = PLC "Di_Ga1.4" AT %I44.3, 1 s
   "Di_Ga2.4" : Bool = PLC "Di_Ga2.4" AT %I44.7, 1 s
   "Kr_1_Work_Run" : Bool = PLC Kr_1_Work.Run, 1 s
   "Kr_2_Work_Run" : Bool = PLC Kr_2_Work.Run, 1 s
   "Kr_1_Work_Step" : Int = PLC Kr_1_Work.Step, 1 s
   "Kr_2_Work_Step" : Int = PLC Kr_2_Work.Step, 1 s
   "Data_GlobalErrorStop" : Bool = PLC Data.GlobalErrorStop, 1 s
   "Data_Equipment_Work" : Bool = PLC Data.Equipment_Work, 1 s
   "WashingWork_DB_Run" : Bool = PLC WashingWork_DB.Run, 1 s
   "Data_Reg_M7_1_Sp" : Real = PLC Data.Reg_M7_1.Sp, 1 s
   "Data_Power_7_2" : Real = PLC Data.Power_7_2, 1 s
   "ViewLine_DB_Line1" : Int = PLC ViewLine_DB.Line1, 1 s
   "ViewLine_DB_Line2" : Int = PLC ViewLine_DB.Line2, 1 s
   "ViewLine_DB_Line3" : Int = PLC ViewLine_DB.Line3, 1 s
   "ViewLine_DB_Line4" : Int = PLC ViewLine_DB.Line4, 1 s
   "ViewLine_DB_Line5" : Int = PLC ViewLine_DB.Line5, 1 s
   "ViewLine_DB_Line6" : Int = PLC ViewLine_DB.Line6, 1 s
   "ViewLine_DB_Line7" : Int = PLC ViewLine_DB.Line7, 1 s
   "ViewLine_DB_Line8" : Int = PLC ViewLine_DB.Line8, 1 s
   "ViewLine_DB_Line9" : Int = PLC ViewLine_DB.Line9, 1 s
   "ViewLine_DB_Line10" : Int = PLC ViewLine_DB.Line10, 1 s
   "ViewLine_DB_Line11" : Int = PLC ViewLine_DB.Line11, 1 s
   "ViewLine_DB_Line12" : Int = PLC ViewLine_DB.Line12, 1 s
   "ViewLine_DB_Line13" : Int = PLC ViewLine_DB.Line13, 1 s
   "ViewLine_DB_Line14" : Int = PLC ViewLine_DB.Line14, 1 s
   "ViewLine_DB_Line15" : Int = PLC ViewLine_DB.Line15, 1 s
   "ViewLine_DB_Line16" : Int = PLC ViewLine_DB.Line16, 1 s
   "ViewLine_DB_Line17" : Int = PLC ViewLine_DB.Line17, 1 s
   "ViewLine_DB_Line18" : Int = PLC ViewLine_DB.Line18, 1 s
   "ViewLine_DB_Line19" : Int = PLC ViewLine_DB.Line19, 1 s
   "ViewLine_DB_Line20" : Int = PLC ViewLine_DB.Line20, 1 s
   "ViewLine_DB_Line21" : Int = PLC ViewLine_DB.Line21, 1 s
   "ViewLine_DB_Line22" : Int = PLC ViewLine_DB.Line22, 1 s
   "ViewLine_DB_Line23" : Int = PLC ViewLine_DB.Line23, 1 s
   "ViewLine_DB_Line24" : Int = PLC ViewLine_DB.Line24, 1 s
   "ViewLine_DB_Line25" : Int = PLC ViewLine_DB.Line25, 1 s
   "Dq_KB1" : Bool = PLC Dq_KB1 AT %Q0.0, 1 s
   "Panel_AreaPointer_DateTimePLC_DateTime" : Date_And_Time = PLC Panel_AreaPointer.DateTimePLC.DateTime AT %DB105.DBX40.0, 1 s
   "Data_ReadyKr2" : Bool = PLC Data.ReadyKr2, 1 s
   "Data_ReadyKr1" : Bool = PLC Data.ReadyKr1, 1 s
   "Data_ReadyCIP" : Bool = PLC Data.ReadyCIP, 1 s
   "Data_Power_7_2_CIP" : Real = PLC Data.Power_7_2_CIP, 1 s
   "WashingWork_DB_Step" : Int = PLC WashingWork_DB.Step, 1 s
   "Data_EnableReady" : Bool = PLC Data.EnableReady, 1 s

discrete alarms
   1: 'Нажата аварийная кнопка', class No Acknowledgement, trigger "Messages" bit 8
   2: 'Напряжение 380В не в норме', class No Acknowledgement, trigger "Messages" bit 9
   3: 'Нет давления воздуха в пневмосистеме', class No Acknowledgement, trigger "Messages" bit 10
   4: 'Верхний аварийный уровень кристализатора №1', class No Acknowledgement, trigger "Messages" bit 11
   5: 'Верхний аварийный уровень кристализатора №2', class No Acknowledgement, trigger "Messages" bit 12
   6: 'Верхний аварийный уровень емкости ледянной воды', class No Acknowledgement, trigger "Messages" bit 13
   7: 'UPS, батарея разряжена', class No Acknowledgement, trigger "Messages" bit 14
   8: 'UPS, батарея неисправна', class No Acknowledgement, trigger "Messages" bit 15
   9: 'Открыт люк 1 кристализатора', class No Acknowledgement, trigger "Messages" bit 0
   10: 'Открыт люк 2 кристализатора', class No Acknowledgement, trigger "Messages" bit 1

text list "cipRegim": 1 'Мойка линии подачи продукта'; 2 'Мойка линии выгрузки продукта'; 3 'Мойка кристализатора №1'; 4 'Мойка кристализатора №2'

text list "Kristal_Regim": 1 'Наполнение'; 2 'Кристализация'; 3 'Выкачка'

text list "on/off": 0 'Отключено'; 1 'Включено'

